CONST robtarget LHP_000:=[[2573.53101,1238.19995,2660.84204],[0.56645757,-0.58473384,0.19941168,-0.54538715],[-1,-1,-1,4],[9E9,9E9,9E9,9E9,9E9,9E9]];
CONST robtarget LHP_005:=[[1933.57397,1076.34998,919.023987],[0.6739808,-0.04561597,0.22679393,-0.70159364],[-1,-1,-1,0],[9E9,9E9,9E9,9E9,9E9,9E9]];
CONST robtarget LHP_010:=[[1910.90503,994.687988,216.904999],[0.7042605,0.08468377,0.09847328,-0.6979605],[-1,-1,-1,0],[9E9,9E9,9E9,9E9,9E9,9E9]];
CONST robtarget LHP_015:=[[1910.89099,994.690002,-385.321991],[0.683501,0.087539785,0.09595496,-0.71830064],[-1,-1,-1,0],[9E9,9E9,9E9,9E9,9E9,9E9]];
CONST robtarget LHP_020:=[[1910.92,803.63,-358.65],[0.683496,0.087554,0.0959515,-0.718305],[-1,-1,-1,0],[9E+09,9E+09,9E+09,9E+09,9E+09,9E+09]];
CONST robtarget LHP_025:=[[1910.97,741.50,-281.66],[0.683494,0.0875455,0.0959486,-0.718307],[-1,-1,-1,0],[9E+09,9E+09,9E+09,9E+09,9E+09,9E+09]];
CONST robtarget LHP_030:=[[1910.91,559.83,-213.69],[0.686476,0.0613746,0.0695917,-0.721208],[-1,-1,-1,0],[9E+09,9E+09,9E+09,9E+09,9E+09,9E+09]];
CONST robtarget LHP_035:=[[1929.33,361.88,-170.13],[0.702471,0.0120548,-0.002609,-0.711605],[-1,0,-1,0],[9E+09,9E+09,9E+09,9E+09,9E+09,9E+09]];
CONST robtarget LHP_040:=[[2007.526,383.55899,-50.7519989],[0.75072795,0.000611088,0.00040383,-0.6606111],[-1,-1,-1,0],[9E9,9E9,9E9,9E9,9E9,9E9]];
CONST robtarget LHP_045:=[[1993.04797,313.046997,-31.7070007],[0.7336252,0.009941696,-0.001285905,-0.67948043],[-1,0,-1,0],[9E9,9E9,9E9,9E9,9E9,9E9]];
CONST robtarget LHP_050:=[[2002.59399,189.292999,-35.1940002],[0.73792726,0.009937888,-0.0012356,-0.67480594],[-1,0,-1,0],[9E9,9E9,9E9,9E9,9E9,9E9]];
CONST robtarget LHP_055:=[[1987.44,-5.82,-69.73],[0.747483,0.000551369,0.000433351,-0.664281],[-1,-1,-1,0],[9E+09,9E+09,9E+09,9E+09,9E+09,9E+09]];
CONST robtarget LHP_060:=[[1929.34,361.89,-170.15],[0.70247,0.0120598,-0.00260928,-0.711607],[-1,0,-1,0],[9E+09,9E+09,9E+09,9E+09,9E+09,9E+09]];
CONST robtarget LHP_065:=[[1910.91,559.85,-213.71],[0.686472,0.0613779,0.0695915,-0.721211],[-1,-1,-1,0],[9E+09,9E+09,9E+09,9E+09,9E+09,9E+09]];
CONST robtarget LHP_070:=[[1769.54,626.69,-228.36],[0.648406,0.063605,0.0595836,-0.756289],[-1,-1,-1,0],[9E+09,9E+09,9E+09,9E+09,9E+09,9E+09]];
CONST robtarget LHP_075:=[[1629.23,373.82,-175.88],[0.60566,0.011527,-0.00436593,-0.795628],[-1,0,-1,0],[9E+09,9E+09,9E+09,9E+09,9E+09,9E+09]];
CONST robtarget LHP_080:=[[1643.37,44.45,-93.67],[0.638426,0.0118697,-0.00343011,-0.769584],[-1,0,-1,0],[9E+09,9E+09,9E+09,9E+09,9E+09,9E+09]];
CONST robtarget LHP_085:=[[1645.79,51.65,-47.78],[0.621544,0.019299,-0.00963586,-0.783082],[-1,0,-1,0],[9E+09,9E+09,9E+09,9E+09,9E+09,9E+09]];
CONST robtarget LHP_090:=[[1652.62,133.53,-52.42],[0.605581,0.0130855,-0.00581803,-0.795655],[-1,0,-1,0],[9E+09,9E+09,9E+09,9E+09,9E+09,9E+09]];
CONST robtarget LHP_095:=[[1617.10803,350.912994,-180.268005],[0.56401443,0.037766688,0.053717423,-0.8231499],[-1,-1,-1,0],[9E9,9E9,9E9,9E9,9E9,9E9]];
CONST robtarget LHP_100:=[[1517.84,635.47,-254.71],[0.565141,-0.00404407,-0.00655324,-0.824958],[-1,0,-1,0],[9E+09,9E+09,9E+09,9E+09,9E+09,9E+09]];
CONST robtarget LHP_105:=[[1647.70,917.36,-357.05],[0.686537,0.012902,0.00966857,-0.726916],[-1,-1,-1,0],[9E+09,9E+09,9E+09,9E+09,9E+09,9E+09]];
CONST robtarget LHP_110:=[[1402.01,954.02,-347.18],[0.618002,-0.00350893,0.00682793,-0.786139],[-1,-1,-1,0],[9E+09,9E+09,9E+09,9E+09,9E+09,9E+09]];
CONST robtarget LHP_115:=[[1380.13,800.38,-344.28],[0.663576,-0.00391562,0.00660285,-0.74807],[-1,-1,-1,0],[9E+09,9E+09,9E+09,9E+09,9E+09,9E+09]];
CONST robtarget LHP_120:=[[1355.05,688.92,-230.68],[0.643458,-0.00406434,0.0069742,-0.765439],[-1,-1,-1,0],[9E+09,9E+09,9E+09,9E+09,9E+09,9E+09]];
CONST robtarget LHP_125:=[[1338.98,616.80,-217.15],[0.641931,-0.00377363,0.00673657,-0.766724],[-1,-1,-1,0],[9E+09,9E+09,9E+09,9E+09,9E+09,9E+09]];
CONST robtarget LHP_130:=[[1328.82,551.60,-198.45],[0.643236,-0.00380631,0.00669098,-0.765629],[-1,-1,-1,0],[9E+09,9E+09,9E+09,9E+09,9E+09,9E+09]];
CONST robtarget LHP_135:=[[1301.19,432.03,-200.08],[0.630965,0.0270779,0.0228783,-0.775001],[-1,-1,-1,0],[9E+09,9E+09,9E+09,9E+09,9E+09,9E+09]];
CONST robtarget LHP_140:=[[1315.22,418.75,-159.95],[0.640955,0.052567,0.0459758,-0.764395],[-1,-1,-1,0],[9E+09,9E+09,9E+09,9E+09,9E+09,9E+09]];
CONST robtarget LHP_145:=[[1314.89,402.01,-58.59],[0.643636,0.0406528,0.0359674,-0.763405],[-1,-1,-1,0],[9E+09,9E+09,9E+09,9E+09,9E+09,9E+09]];
CONST robtarget LHP_150:=[[1314.89,402.00,-58.59],[0.64363700,0.04065100,0.0359677,-0.7634040],[-1,-1,-1,0],[9E+09,9E+09,9E+09,9E+09,9E+09,9E+09]];
CONST robtarget LHP_155:=[[1315.25,418.75,-159.98],[0.640959,0.05257270,0.04597540,-0.7643910],[-1,-1,-1,0],[9E+09,9E+09,9E+09,9E+09,9E+09,9E+09]];
CONST robtarget LHP_160:=[[1301.20,432.03,-200.09],[0.630966,0.0270787,0.0228773,-0.775],[-1,-1,-1,0],[9E+09,9E+09,9E+09,9E+09,9E+09,9E+09]];
CONST robtarget LHP_165:=[[1328.84,551.60,-198.48],[0.643767,-0.00379566,0.00669219,-0.765183],[-1,-1,-1,0],[9E+09,9E+09,9E+09,9E+09,9E+09,9E+09]];
CONST robtarget LHP_170:=[[1356.81,663.69,-214.66],[0.64609,-0.00377796,0.00670482,-0.7632220],[-1,-1,-1,0],[9E+09,9E+09,9E+09,9E+09,9E+09,9E+09]];
CONST robtarget LHP_175:=[[1392.09,854.35,-337.39],[0.646086,-0.00378978,0.00670626,-0.763226],[-1,-1,-1,0],[9E+09,9E+09,9E+09,9E+09,9E+09,9E+09]];
CONST robtarget LHP_180:=[[1392.10,915.32,-339.98],[0.646085,-0.00379686,0.00670629,-0.763227],[-1,-1,-1,0],[9E+09,9E+09,9E+09,9E+09,9E+09,9E+09]];
CONST robtarget LHP_185:=[[1392.13,915.34,-336.92],[0.646086,-0.00378783,0.00670572,-0.763226],[-1,-1,-1,0],[9E+09,9E+09,9E+09,9E+09,9E+09,9E+09]];
CONST robtarget LHP_190:=[[1777.10,396.39,-174.51],[0.778298,0.00338922,-0.00251072,-0.62788],[-1,0,-1,0],[9E+09,9E+09,9E+09,9E+09,9E+09,9E+09]];
CONST robtarget LHP_195:=[[1816.72,397.75,-147.92],[0.816486,0.00152322,-0.000785194,-0.577362],[-1,0,-1,0],[9E+09,9E+09,9E+09,9E+09,9E+09,9E+09]];
CONST robtarget LHP_200:=[[1816.69,397.74,-147.92],[0.816487,0.00151316,-0.000780112,-0.577362],[-1,0,-1,0],[9E+09,9E+09,9E+09,9E+09,9E+09,9E+09]];
CONST robtarget LHP_205:=[[1684.96,400.28,-45.26],[0.59824,-0.000475336,-0.0146536,-0.801183],[-1,0,-1,0],[9E+09,9E+09,9E+09,9E+09,9E+09,9E+09]];
CONST robtarget LHP_210:=[[1517.37,845.68,-347.51],[0.603966,0.0765094,0.0409368,-0.792272],[-1,-1,-1,0],[9E+09,9E+09,9E+09,9E+09,9E+09,9E+09]];
CONST robtarget LHP_215:=[[1614.81,303.29,-114.97],[0.595541,4.37463E-06,7.52158E-05,-0.803325],[-1,-1,-1,0],[9E+09,9E+09,9E+09,9E+09,9E+09,9E+09]];
CONST robtarget LHP_220:=[[1496.10,381.00,-140.90],[0.501832,0.0142883,0.0357857,-0.864106],[-1,-1,-1,0],[9E+09,9E+09,9E+09,9E+09,9E+09,9E+09]];
CONST robtarget LHP_225:=[[1496.16,381.04,-179.37],[0.501836,0.0143261,0.0358019,-0.864103],[-1,-1,-1,0],[9E+09,9E+09,9E+09,9E+09,9E+09,9E+09]];
CONST robtarget LHP_230:=[[1517.37,556.59,-186.35],[0.545787,0.0365786,0.0545327,-0.835347],[-1,-1,-1,0],[9E+09,9E+09,9E+09,9E+09,9E+09,9E+09]];
CONST robtarget LHP_235:=[[1529.66,619.50,-150.47],[0.565262,-0.000227126,0.000165536,-0.824912],[-1,-1,-1,0],[9E+09,9E+09,9E+09,9E+09,9E+09,9E+09]];
CONST robtarget LHP_240:=[[1558.44,796.09,-349.49],[0.583985,0.0684408,0.0319346,-0.808244],[-1,-1,-1,0],[9E+09,9E+09,9E+09,9E+09,9E+09,9E+09]];
CONST robtarget LHP_245:=[[1477.93,985.71,-357.82],[0.551096,0.0897034,0.0519627,-0.827978],[-1,-1,-1,0],[9E+09,9E+09,9E+09,9E+09,9E+09,9E+09]];
CONST robtarget LHP_250:=[[807.86,896.51,-348.98],[0.475989,-0.019585,0.0486327,-0.877887],[-1,-1,-1,0],[9E+09,9E+09,9E+09,9E+09,9E+09,9E+09]];
CONST robtarget LHP_255:=[[807.84,813.89,-348.98],[0.47599,-0.0195894,0.0486332,-0.877887],[-1,-1,-1,0],[9E+09,9E+09,9E+09,9E+09,9E+09,9E+09]];
CONST robtarget LHP_260:=[[798.625,757.187988,-251.093002],[0.47488588,-0.019798715,0.048936285,-0.8784627],[-1,-1,-1,0],[9E9,9E9,9E9,9E9,9E9,9E9]];
CONST robtarget LHP_265:=[[687.672974,377.386993,-182.552002],[0.5034063,-0.04137853,0.03811411,-0.8622165],[-1,-1,-1,0],[9E9,9E9,9E9,9E9,9E9,9E9]];
CONST robtarget LHP_270:=[[796.06,403.61,2.12],[0.54967,-0.0809587,0.0198978,-0.831212],[-1,-1,-1,0],[9E+09,9E+09,9E+09,9E+09,9E+09,9E+09]];
CONST robtarget LHP_275:=[[951.56,404.05,-36.64],[0.666081,-0.0483269,0.018538,-0.744081],[-1,-1,-1,0],[9E+09,9E+09,9E+09,9E+09,9E+09,9E+09]];
CONST robtarget LHP_280:=[[1053.17,384.08,-147.35],[0.741703,0.0276666,0.0554714,-0.667858],[-1,-1,-1,0],[9E+09,9E+09,9E+09,9E+09,9E+09,9E+09]];
CONST robtarget LHP_285:=[[1117.00,437.68,-186.63],[0.764604,0.0628167,0.0737039,-0.637183],[-1,-1,-1,0],[9E+09,9E+09,9E+09,9E+09,9E+09,9E+09]];
CONST robtarget LHP_290:=[[1206.43,437.70,-186.66],[0.808318,0.0679399,0.0690137,-0.580726],[-1,-1,-1,0],[9E+09,9E+09,9E+09,9E+09,9E+09,9E+09]];
CONST robtarget LHP_295:=[[1254.01,306.17,-147.47],[0.819239,0.0692406,0.0677067,-0.565215],[-1,-1,-1,0],[9E+09,9E+09,9E+09,9E+09,9E+09,9E+09]];
CONST robtarget LHP_300:=[[1294.76,251.64,-118.31],[0.839473,0.0657832,0.0563212,-0.536456],[-1,-1,-1,0],[9E+09,9E+09,9E+09,9E+09,9E+09,9E+09]];
CONST robtarget LHP_305:=[[1302.68,268.91,-77.08],[0.850295,0.0194976,0.0312356,-0.525017],[-1,-1,-1,0],[9E+09,9E+09,9E+09,9E+09,9E+09,9E+09]];
CONST robtarget LHP_310:=[[1302.67,268.92,-77.09],[0.850295,0.0194964,0.0312402,-0.525016],[-1,-1,-1,0],[9E+09,9E+09,9E+09,9E+09,9E+09,9E+09]];
CONST robtarget LHP_315:=[[1294.76,251.64,-118.31],[0.839473,0.0657839,0.0563209,-0.536456],[-1,-1,-1,0],[9E+09,9E+09,9E+09,9E+09,9E+09,9E+09]];
CONST robtarget LHP_320:=[[1254.01,306.17,-147.47],[0.819239,0.0692405,0.0677067,-0.565215],[-1,-1,-1,0],[9E+09,9E+09,9E+09,9E+09,9E+09,9E+09]];
CONST robtarget LHP_325:=[[1206.43,437.70,-186.66],[0.808318,0.0679399,0.0690137,-0.580726],[-1,-1,-1,0],[9E+09,9E+09,9E+09,9E+09,9E+09,9E+09]];
CONST robtarget LHP_330:=[[1117.00,437.68,-186.63],[0.764604,0.0628167,0.0737039,-0.637183],[-1,-1,-1,0],[9E+09,9E+09,9E+09,9E+09,9E+09,9E+09]];
CONST robtarget LHP_335:=[[1116.98,404.12,-155.12],[0.767929,0.0632076,0.0733697,-0.633172],[-1,-1,-1,0],[9E+09,9E+09,9E+09,9E+09,9E+09,9E+09]];
CONST robtarget LHP_340:=[[1116.98,404.12,-77.86],[0.763388,0.0288222,0.0341692,-0.644392],[-1,-1,-1,0],[9E+09,9E+09,9E+09,9E+09,9E+09,9E+09]];
CONST robtarget LHP_345:=[[951.56,404.05,-36.63],[0.666079,-0.0483271,0.018537,-0.744083],[-1,-1,-1,0],[9E+09,9E+09,9E+09,9E+09,9E+09,9E+09]];
CONST robtarget LHP_350:=[[863.42,413.34,0.81],[0.590286,-0.0726155,0.0279581,-0.803435],[-1,-1,-1,0],[9E+09,9E+09,9E+09,9E+09,9E+09,9E+09]];
CONST robtarget LHP_355:=[[687.66803,377.371002,-182.531006],[0.5034058,-0.04138605,0.0381097,-0.8622166],[-1,-1,-1,0],[9E9,9E9,9E9,9E9,9E9,9E9]];
CONST robtarget LHP_360:=[[798.580994,757.198975,-251.070007],[0.47486982,-0.019813199,0.04892835,-0.8784715],[-1,-1,-1,0],[9E9,9E9,9E9,9E9,9E9,9E9]];
CONST robtarget LHP_365:=[[961.40,981.11,-456.97],[0.440335,0.0935079,0.0750373,-0.889792],[-1,-1,-1,0],[9E+09,9E+09,9E+09,9E+09,9E+09,9E+09]];
CONST robtarget LHP_370:=[[1477.90,985.72,-357.83],[0.558631,0.0901634,0.0511329,-0.822914],[-1,-1,-1,0],[9E+09,9E+09,9E+09,9E+09,9E+09,9E+09]];
CONST robtarget LHP_375:=[[1538.22,786.86,-339.64],[0.544053,0.0691445,0.0535195,-0.834482],[-1,-1,-1,0],[9E+09,9E+09,9E+09,9E+09,9E+09,9E+09]];
CONST robtarget LHP_380:=[[1502.92,670.32,-266.02],[0.529086,0.0479959,0.0506422,-0.845695],[-1,-1,-1,0],[9E+09,9E+09,9E+09,9E+09,9E+09,9E+09]];
CONST robtarget LHP_385:=[[1496.13,395.81,-167.92],[0.501832,0.0142997,0.0357903,-0.864106],[-1,-1,-1,0],[9E+09,9E+09,9E+09,9E+09,9E+09,9E+09]];
CONST robtarget LHP_390:=[[1515.01,305.29,-41.45],[0.500229,-6.95049E-05,2.93455E-05,-0.865893],[-1,-1,-1,0],[9E+09,9E+09,9E+09,9E+09,9E+09,9E+09]];
CONST robtarget LHP_395:=[[1371.85706,156.694901,-47.4344292],[0.4850808,-0.004593692,-0.00611278,-0.8744359],[-1,0,-1,0],[9E9,9E9,9E9,9E9,9E9,9E9]];
CONST robtarget LHP_400:=[[1371.81006,156.684998,-41.7470016],[0.48507392,-0.004586132,-0.006106427,-0.8744398],[-1,0,-1,0],[9E9,9E9,9E9,9E9,9E9,9E9]];
CONST robtarget LHP_405:=[[1492.72,315.84,-138.22],[0.571745,-0.00395765,-0.00657566,-0.820395],[-1,0,-1,0],[9E+09,9E+09,9E+09,9E+09,9E+09,9E+09]];
CONST robtarget LHP_410:=[[1568.64,542.95,-202.94],[0.571744,-0.00395848,-0.00658119,-0.820396],[-1,0,-1,0],[9E+09,9E+09,9E+09,9E+09,9E+09,9E+09]];
CONST robtarget LHP_415:=[[1568.58,736.45,-284.14],[0.571745,-0.00397095,-0.00657964,-0.820396],[-1,0,-1,0],[9E+09,9E+09,9E+09,9E+09,9E+09,9E+09]];
CONST robtarget LHP_420:=[[1508.30,917.00,-395.22],[0.556499,0.0508994,0.0317793,-0.828678],[-1,-1,-1,0],[9E+09,9E+09,9E+09,9E+09,9E+09,9E+09]];
CONST robtarget LHP_425:=[[1495.25,987.39,-357.83],[0.551104,0.0895725,0.0518729,-0.827992],[-1,-1,-1,0],[9E+09,9E+09,9E+09,9E+09,9E+09,9E+09]];
CONST robtarget LHP_430:=[[1328.35,635.44,-278.20],[0.501405,0.0212305,0.11734,-0.856956],[-1,-1,0,0],[9E+09,9E+09,9E+09,9E+09,9E+09,9E+09]];
CONST robtarget LHP_435:=[[1126.70,526.89,-238.13],[0.384755,0.0646485,0.107006,-0.914513],[-1,-1,0,0],[9E+09,9E+09,9E+09,9E+09,9E+09,9E+09]];
CONST robtarget LHP_440:=[[1126.70,526.87,-238.14],[0.384757,0.0646487,0.107006,-0.914512],[-1,-1,0,0],[9E+09,9E+09,9E+09,9E+09,9E+09,9E+09]];
CONST robtarget LHP_445:=[[1328.35,635.43,-278.21],[0.501406,0.0212292,0.11734,-0.856956],[-1,-1,0,0],[9E+09,9E+09,9E+09,9E+09,9E+09,9E+09]];
CONST robtarget LHP_450:=[[1495.26,987.39,-357.84],[0.551103,0.0895724,0.0518701,-0.827993],[-1,-1,-1,0],[9E+09,9E+09,9E+09,9E+09,9E+09,9E+09]];
CONST robtarget LHP_455:=[[1606.25,805.30,-336.47],[0.591189,0.0705667,0.0504833,-0.801852],[-1,-1,-1,0],[9E+09,9E+09,9E+09,9E+09,9E+09,9E+09]];
CONST robtarget LHP_460:=[[1846.21,646.41,-266.45],[0.66313,0.055392,0.0578373,-0.744207],[-1,-1,-1,0],[9E+09,9E+09,9E+09,9E+09,9E+09,9E+09]];
CONST robtarget LHP_465:=[[1831.93,634.62,-78.38],[0.625946,0.00957367,0.0100376,-0.779743],[-1,-1,-1,0],[9E+09,9E+09,9E+09,9E+09,9E+09,9E+09]];
CONST robtarget LHP_470:=[[1778.25,512.89,-42.92],[0.553639,0.000122695,-2.9028E-05,-0.832757],[-1,-1,-1,0],[9E+09,9E+09,9E+09,9E+09,9E+09,9E+09]];
CONST robtarget LHP_475:=[[1581.22,548.75,-125.86],[0.508525,0.0149425,0.00198371,-0.860915],[-1,0,-1,0],[9E+09,9E+09,9E+09,9E+09,9E+09,9E+09]];
CONST robtarget LHP_480:=[[1526.71,530.36,-111.44],[0.495097,0.0157343,0.00230728,-0.868692],[-1,0,-1,0],[9E+09,9E+09,9E+09,9E+09,9E+09,9E+09]];
CONST robtarget LHP_485:=[[1496.52905,533.620972,-169.427002],[0.5015252,0.014323151,0.035049833,-0.8643141],[-1,-1,-1,0],[9E9,9E9,9E9,9E9,9E9,9E9]];
CONST robtarget LHP_490:=[[1628.88,359.00,-167.42],[0.509965,0.00587853,-0.00326077,-0.860169],[-1,0,-1,0],[9E+09,9E+09,9E+09,9E+09,9E+09,9E+09]];
CONST robtarget LHP_495:=[[1653.10,363.04,-167.43],[0.50985,0.0307676,0.0114918,-0.859636],[-1,0,-1,0],[9E+09,9E+09,9E+09,9E+09,9E+09,9E+09]];
CONST robtarget LHP_500:=[[1734.14,581.56,-229.81],[0.51369,0.0926739,0.046858,-0.851668],[-1,-1,-1,0],[9E+09,9E+09,9E+09,9E+09,9E+09,9E+09]];
CONST robtarget LHP_505:=[[1850.77,754.32,-287.10],[0.562259,0.138379,0.0973397,-0.809469],[-1,-1,-1,0],[9E+09,9E+09,9E+09,9E+09,9E+09,9E+09]];
CONST robtarget LHP_510:=[[1850.71,883.30,-361.37],[0.589549,0.148661,0.155296,-0.778598],[-1,-1,-1,0],[9E+09,9E+09,9E+09,9E+09,9E+09,9E+09]];
CONST robtarget LHP_515:=[[1850.60,911.16,-304.76],[0.610795,0.143869,0.202267,-0.751877],[-1,-1,-1,0],[9E+09,9E+09,9E+09,9E+09,9E+09,9E+09]];
CONST robtarget LHP_520:=[[1845.93,938.54,-187.19],[0.617535,0.126482,0.223985,-0.743292],[-1,-1,-1,0],[9E+09,9E+09,9E+09,9E+09,9E+09,9E+09]];
CONST robtarget LHP_525:=[[1839.91,764.25,251.37],[0.609113,0.0794277,0.135403,-0.777392],[-1,-1,-1,0],[9E+09,9E+09,9E+09,9E+09,9E+09,9E+09]];
CONST robtarget LHP_530:=[[1951.53,815.35,1215.32],[0.610126,-0.0704393,-0.00824645,-0.789124],[-1,0,-1,0],[9E+09,9E+09,9E+09,9E+09,9E+09,9E+09]];
CONST robtarget LHP_535:=[[2438.93,960.39,2235.39],[0.671457,-0.189483,-0.125804,-0.705277],[-1,0,-1,0],[9E+09,9E+09,9E+09,9E+09,9E+09,9E+09]];
!provisorische Punkte fuer SP-Versetzung in Zone2
CONST robtarget LHP_605:=[[1647.70,917.36,-357.05],[0.686537,0.012902,0.00966857,-0.726916],[-1,-1,-1,0],[9E+09,9E+09,9E+09,9E+09,9E+09,9E+09]];
CONST robtarget LHP_610:=[[1610.73,498.12,-174.33],[0.637115,0.00115243,-0.000308458,-0.770768],[-1,0,-1,0],[9E+09,9E+09,9E+09,9E+09,9E+09,9E+09]];
CONST robtarget LHP_620:=[[1777.10,396.39,-174.52],[0.764298,0.00344259,-0.00243544,-0.644849],[-1,0,-1,0],[9E+09,9E+09,9E+09,9E+09,9E+09,9E+09]];
CONST robtarget LHP_625:=[[1816.72,397.75,-147.92],[0.816486,0.00152322,-0.000785194,-0.577362],[-1,0,-1,0],[9E+09,9E+09,9E+09,9E+09,9E+09,9E+09]];
CONST robtarget LHP_630:=[[1816.69,397.74,-147.92],[0.816487,0.00151316,-0.000780112,-0.577362],[-1,0,-1,0],[9E+09,9E+09,9E+09,9E+09,9E+09,9E+09]];
CONST robtarget LHP_635:=[[1517.21,788.33,-328.51],[0.603967,0.0765054,0.0409354,-0.792272],[-1,-1,-1,0],[9E+09,9E+09,9E+09,9E+09,9E+09,9E+09]];
CONST robtarget LHP_600:=[[1990.20,974.03,1486.76],[0.667207,-0.21865,0.214527,-0.678974],[-1,-1,-1,0],[9E+09,9E+09,9E+09,9E+09,9E+09,9E+09]];
! ------------------------------------------------------------
! Unterprogramm:
! Stand
! Daimler AG - Werk Ludwigsfelde
! ------------------------------------------------------------
! ************************************************************
! Kommentar: Achtung
! automatisch generiert!!!!!!!!!!!!!!!!!!
! ************************************************************

! Robotername: 1606R04
! Anlagenbezeichn: Linie 16 Stations-Nr: 1606
! Stand / Version: 04.08.2009 / 1.1
! Name Bearbeiter: Karmann
! Applikationssteuerung: Punktschweissen
! Baumuster: FHL T1 R2


INIT_SW_BASE;

WKZ_1_AUFNEHMEN;

MoveJ ToolHome1,vSchnell,fine,nomtcp1;

MoveJ LHP_000,vSchnell,fine,nomtcp1\WObj:=BS_1606_1A;

Vorhub\auf;

ABL 2\ABL_WAIT;
ABL 10\ABL_SET;

!1606R04_1606R06
KOLLISION_ZONE 2\Anfrage;
!1606R04_1606R06
KOLLISION_ZONE 7\Anfrage;
!1606R04_1606R06
KOLLISION_ZONE 9\Anfrage;

MoveJ LHP_600, vSchnell, fine, nomtcp1\WObj:=BS_1606_1A;

!
! robic dojazd
!
WaitUntil FALSE;

MoveJ LHP_165,vSchnell,z100,nomtcp1\WObj:=BS_1606_1A;
MoveJ LHP_160,vSchnell,z1,nomtcp1\WObj:=BS_1606_1A;
MoveJ LHP_155,vSchnell,z1,nomtcp1\WObj:=BS_1606_1A;
MoveJ LHP_150,vSchnell,z1,nomtcp1\WObj:=BS_1606_1A;

SpotL G0216190478BP20\VFO:=210,vSpot,nomtcp1\WObj:=BS_1606_1A;
SpotL G0216190582BP20\VFO:=210,vSpot,nomtcp1\WObj:=BS_1606_1A;

MoveJ LHP_120,vSchnell,z100,nomtcp1\WObj:=BS_1606_1A;
MoveJ LHP_125,vSchnell,z100,nomtcp1\WObj:=BS_1606_1A;

SpotL G0216190492BP20\VFO:=210\Vorhub_Auf,vSpot,nomtcp1\WObj:=BS_1606_1A;

KOLLISION_ZONE 2\Freigabe;

!
! zrobic dojazd
!
WaitUntil FALSE;

MoveJ LHP_480,vSchnell,z100,nomtcp1\WObj:=BS_1606_1A;

SpotL G0216190576BP20\VFO:=210,vSpot,nomtcp1\WObj:=BS_1606_1A;
SpotL G0213198812BP20\VFO:=210\Vorhub_Auf,vSpot,nomtcp1\WObj:=BS_1606_1A;

MoveJ LHP_485,vSchnell,z100,nomtcp1\WObj:=BS_1606_1A;

!
! zrobic dojazd
!
WaitUntil FALSE;

SpotL G0213198810BP20\VFO:=210,vSpot,nomtcp1\WObj:=BS_1606_1A;
SpotL G0213198808BP20\VFO:=210,vSpot,nomtcp1\WObj:=BS_1606_1A;
SpotL G0216021648BP20\VFO:=210,vSpot,nomtcp1\WObj:=BS_1606_1A;
SpotL G0216021650BP20\VFO:=210,vSpot,nomtcp1\WObj:=BS_1606_1A;

MoveJ LHP_470,vSchnell,fine,nomtcp1\WObj:=BS_1606_1A;

SpotL G0216021652BP20\VFO:=210,vSpot,nomtcp1\WObj:=BS_1606_1A;

!
! zrobic dojazd
!
WaitUntil FALSE;

MoveJ LHP_620,vSchnell,z100,nomtcp1\WObj:=BS_1606_1A;
MoveJ LHP_625,vSchnell,z100,nomtcp1\WObj:=BS_1606_1A;

SpotL G0216021802BP20\VFO:=210\Vorhub_Auf,vSpot,nomtcp1\WObj:=BS_1606_1A;

MoveJ LHP_630,vSchnell,z100,nomtcp1\WObj:=BS_1606_1A;

!
! zrobic dojazd
!
WaitUntil FALSE;

MoveJ LHP_025,vSchnell,z100,nomtcp1\WObj:=BS_1606_1A;
MoveJ LHP_030,vSchnell,z100,nomtcp1\WObj:=BS_1606_1A;
MoveJ LHP_035,vSchnell,z100,nomtcp1\WObj:=BS_1606_1A;

SpotL G0216021800BP20\VFO:=210,vSpot,nomtcp1\WObj:=BS_1606_1A;
SpotL G0216021798BP20\VFO:=210\Vorhub_Auf,vSpot,nomtcp1\WObj:=BS_1606_1A;

!
! zrobic dojazd
!
WaitUntil FALSE;

SpotL G0216021654BP20\VFO:=210,vSpot,nomtcp1\WObj:=BS_1606_1A;
SpotL G0216190440BP20\VFO:=210,vSpot,nomtcp1\WObj:=BS_1606_1A;
SpotL G0216190438BP20\VFO:=210,vSpot,nomtcp1\WObj:=BS_1606_1A;

MoveJ LHP_455,vSchnell,z100,nomtcp1\WObj:=BS_1606_1A;
MoveJ LHP_460,vSchnell,z100,nomtcp1\WObj:=BS_1606_1A;
MoveJ LHP_465,vSchnell,z100,nomtcp1\WObj:=BS_1606_1A;

SpotL G0216190436BP20\VFO:=210\Vorhub_Auf,vSpot,nomtcp1\WObj:=BS_1606_1A;

!
! zrobic dojazd
!
WaitUntil FALSE;

MoveJ LHP_475,vSchnell,z100,nomtcp1\WObj:=BS_1606_1A;

SpotL G0216190434BP20\VFO:=210,vSpot,nomtcp1\WObj:=BS_1606_1A;
SpotL G0216190432BP20\VFO:=210,vSpot,nomtcp1\WObj:=BS_1606_1A;
SpotL G0216190430BP20\VFO:=210,vSpot,nomtcp1\WObj:=BS_1606_1A;

MoveJ LHP_450,vSchnell,z100,nomtcp1\WObj:=BS_1606_1A;

SpotL G0216190428BP20\VFO:=210\Vorhub_Auf,vSpot,nomtcp1\WObj:=BS_1606_1A;

!
! zrobic dojazd
!
WaitUntil FALSE;

MoveJ LHP_230,vSchnell,z100,nomtcp1\WObj:=BS_1606_1A;

SpotL G0216190446BP20\VFO:=210\Vorhub_Auf,vSpot,nomtcp1\WObj:=BS_1606_1A;

MoveJ LHP_235,vSchnell,z100,nomtcp1\WObj:=BS_1606_1A;
MoveJ LHP_610,vSchnell,fine,nomtcp1\WObj:=BS_1606_1A;

!
! zrobic dojazd
!
WaitUntil FALSE;

MoveJ LHP_250,vSchnell,fine,nomtcp1\WObj:=BS_1606_1A;

!1606R04_1606R06
KOLLISION_ZONE 1\Anfrage;
!1606R04_1606R06
KOLLISION_ZONE 6\Anfrage;

MoveJ LHP_255,vSchnell,z100,nomtcp1\WObj:=BS_1606_1A;
MoveJ LHP_260,vSchnell,z100,nomtcp1\WObj:=BS_1606_1A;
MoveJ LHP_265,vSchnell,z100,nomtcp1\WObj:=BS_1606_1A;
MoveJ LHP_270,vSchnell,z100,nomtcp1\WObj:=BS_1606_1A;
MoveJ LHP_275,vSchnell,z100,nomtcp1\WObj:=BS_1606_1A;
MoveJ LHP_280,vSchnell,z100,nomtcp1\WObj:=BS_1606_1A;
MoveL LHP_285,vSchnell,z5,nomtcp1\WObj:=BS_1606_1A;
MoveL LHP_290,vSchnell,z5,nomtcp1\WObj:=BS_1606_1A;
MoveL LHP_295,vSchnell,z5,nomtcp1\WObj:=BS_1606_1A;
MoveL LHP_300,vSchnell,z5,nomtcp1\WObj:=BS_1606_1A;
MoveL LHP_305,vSchnell,z5,nomtcp1\WObj:=BS_1606_1A;

SpotL G0216190480BP20\VFO:=210\Vorhub_Auf, vSpot, nomtcp1\WObj:=BS_1606_1A;

MoveL LHP_310,vSchnell,z5,nomtcp1\WObj:=BS_1606_1A;
MoveL LHP_315,vSchnell,z5,nomtcp1\WObj:=BS_1606_1A;
MoveL LHP_320,vSchnell,z5,nomtcp1\WObj:=BS_1606_1A;
MoveL LHP_325,vSchnell,z5,nomtcp1\WObj:=BS_1606_1A;
MoveL LHP_330,vSchnell,z5,nomtcp1\WObj:=BS_1606_1A;
MoveL LHP_335,vSchnell,z5,nomtcp1\WObj:=BS_1606_1A;
MoveL LHP_340,vSchnell,z5,nomtcp1\WObj:=BS_1606_1A;

SpotL G0216022394BP20\VFO:=210\Vorhub_Auf,vSpot,nomtcp1\WObj:=BS_1606_1A;

MoveJ LHP_345,vSchnell,fine,nomtcp1\WObj:=BS_1606_1A;
MoveJ LHP_350,vSchnell,z100,nomtcp1\WObj:=BS_1606_1A;

SpotL G0216022386BP20\VFO:=210,vSpot,nomtcp1\WObj:=BS_1606_1A;

!1606R04_1606R06
KOLLISION_ZONE 6\Freigabe;

SpotL G0216047033BP20\VFO:=210,vSpot,nomtcp1\WObj:=BS_1606_1A;
SpotL G0216047032BP20\VFO:=210\Vorhub_Auf,vSpot,nomtcp1\WObj:=BS_1606_1A;

MoveJ LHP_355,vSchnell,z100,nomtcp1\WObj:=BS_1606_1A;
MoveJ LHP_360,vSchnell,z100,nomtcp1\WObj:=BS_1606_1A;
MoveJ LHP_365,vSchnell,z100,nomtcp1\WObj:=BS_1606_1A;
MoveJ LHP_370,vSchnell,z100,nomtcp1\WObj:=BS_1606_1A;
!
! zrobic dojazd
!
WaitUntil FALSE;

MoveJ LHP_420,vSchnell,z100,nomtcp1\WObj:=BS_1606_1A;
MoveJ LHP_425,vSchnell,z100,nomtcp1\WObj:=BS_1606_1A;
MoveJ LHP_430,vSchnell,z100,nomtcp1\WObj:=BS_1606_1A;
MoveJ LHP_435,vSchnell,z100,nomtcp1\WObj:=BS_1606_1A;

SpotL G0216047028BP20\VFO:=210,vSpot,nomtcp1\WObj:=BS_1606_1A;
SpotL G0216047029BP20\VFO:=210,vSpot,nomtcp1\WObj:=BS_1606_1A;
SpotL G0216022368BP20\VFO:=210,vSpot,nomtcp1\WObj:=BS_1606_1A;
SpotL G0216022370BP20\VFO:=210\Vorhub_Auf,vSpot,nomtcp1\WObj:=BS_1606_1A;

MoveJ LHP_440,vSchnell,z100,nomtcp1\WObj:=BS_1606_1A;

!
! zrobic dojazd
!
waituntil FALSE;

MoveJ LHP_040,vSchnell,z100,nomtcp1\WObj:=BS_1606_1A;

SpotL G0216190516BP20\VFO:=210,vSpot,nomtcp1\WObj:=BS_1606_1A;

MoveJ LHP_045,vSchnell,z100,nomtcp1\WObj:=BS_1606_1A;

KOLLISION_ZONE 1\Freigabe;
KOLLISION_ZONE 7\Freigabe;
KOLLISION_ZONE 8\Anfrage;

SpotL G0216190518BP20\VFO:=210,vSpot,nomtcp1\WObj:=BS_1606_1A;
SpotL G0216190520BP20\VFO:=210,vSpot,nomtcp1\WObj:=BS_1606_1A;

MoveJ LHP_050,vSchnell,z100,nomtcp1\WObj:=BS_1606_1A;

SpotL G0216190522BP20\VFO:=210,vSpot,nomtcp1\WObj:=BS_1606_1A;
SpotL G0216190524BP20\VFO:=210,vSpot,nomtcp1\WObj:=BS_1606_1A;

!1606R04_1606R03
KOLLISION_ZONE 4\Anfrage;

SpotL G0216190526BP20\VFO:=210,vSpot,nomtcp1\WObj:=BS_1606_1A;
SpotL G0216190528BP20\VFO:=210\Vorhub_Auf, vSpot, nomtcp1\WObj:=BS_1606_1A;

MoveJ LHP_055,vSchnell,z100,nomtcp1\WObj:=BS_1606_1A;
MoveJ LHP_060,vSchnell,z100,nomtcp1\WObj:=BS_1606_1A;
MoveJ LHP_065,vSchnell,z100,nomtcp1\WObj:=BS_1606_1A;
MoveJ LHP_070,vSchnell,z100,nomtcp1\WObj:=BS_1606_1A;
MoveJ LHP_075,vSchnell,z100,nomtcp1\WObj:=BS_1606_1A;
MoveJ LHP_080,vSchnell,z100,nomtcp1\WObj:=BS_1606_1A;

SpotL G0216190508BP20\VFO:=210,vSpot,nomtcp1\WObj:=BS_1606_1A;

MoveJ LHP_085,vSchnell,z100,nomtcp1\WObj:=BS_1606_1A;
MoveJ LHP_090,vSchnell,z100,nomtcp1\WObj:=BS_1606_1A;

SpotL G0216190500BP20\VFO:=210,vSpot,nomtcp1\WObj:=BS_1606_1A;
SpotL G0216190506BP20\VFO:=210,vSpot,nomtcp1\WObj:=BS_1606_1A;

!
! zrobic dojazd
!
WaitUntil FALSE;

MoveJ LHP_385,vSchnell,z100,nomtcp1\WObj:=BS_1606_1A;
MoveJ LHP_390,vSchnell,fine,nomtcp1\WObj:=BS_1606_1A;

!1606R04_1606R06
KOLLISION_ZONE 7\Freigabe;

SpotL G0216190498BP20\VFO:=210,vSpot,nomtcp1\WObj:=BS_1606_1A;

MoveJ LHP_395,vSchnell,z100,nomtcp1\WObj:=BS_1606_1A;

SpotL G0216190488BP20\VFO:=210,vSpot,nomtcp1\WObj:=BS_1606_1A;

MoveJ LHP_400,vSchnell,z100,nomtcp1\WObj:=BS_1606_1A;

SpotL G0216190496BP20\VFO:=210,vSpot,nomtcp1\WObj:=BS_1606_1A;
SpotL G0216190494BP20\VFO:=210\Vorhub_Auf,vSpot,nomtcp1\WObj:=BS_1606_1A;

MoveJ LHP_405,vSchnell,z100,nomtcp1\WObj:=BS_1606_1A;

!
! zrobic dojazd
!
WaitUntil FALSE;

SpotL G0216190502BP20\VFO:=210\Vorhub_Auf,vSpot,nomtcp1\WObj:=BS_1606_1A;

MoveJ LHP_215, vSchnell, z100, nomtcp1\WObj:=BS_1606_1A;
MoveJ LHP_220, vSchnell, z100, nomtcp1\WObj:=BS_1606_1A;

KOLLISION_ZONE 8\Freigabe;

SpotL G0213198814BP20\VFO:=210\Vorhub_Auf,vSpot,nomtcp1\WObj:=BS_1606_1A;

MoveJ LHP_225,vSchnell,z100,nomtcp1\WObj:=BS_1606_1A;

!
! zrobic dojazd
!
WaitUntil FALSE;

SpotL G0213198816BP20\VFO:=210,vSpot,nomtcp1\WObj:=BS_1606_1A;
SpotL G0213198818BP20\VFO:=210\Vorhub_Auf,vSpot,nomtcp1\WObj:=BS_1606_1A;

MoveJ LHP_495,vSchnell,z100,nomtcp1\WObj:=BS_1606_1A;
MoveJ LHP_500,vSchnell,z10,nomtcp1\WObj:=BS_1606_1A;
MoveJ LHP_505,vSchnell,z5,nomtcp1\WObj:=BS_1606_1A;

!
! zrobic dojazd
!
WaitUntil FALSE;

MoveJ LHP_205,vSchnell,z100,nomtcp1\WObj:=BS_1606_1A;

SpotL G0216021806BP20\VFO:=210,vSpot,nomtcp1\WObj:=BS_1606_1A;
SpotL G0216021804BP20\VFO:=210\Vorhub_Auf,vSpot,nomtcp1\WObj:=BS_1606_1A;


!1606R04_1606R06
KOLLISION_ZONE 1\Freigabe;

MoveJ LHP_535, vSchnell, z100, nomtcp1\WObj:=BS_1606_1A;

MoveJ ToolHome1,vSchnell,fine,nomtcp1;


ABL 254\ABL_WAIT;
ABL 255\ABL_SET;

!1606R04_1606R06
KOLLISION_ZONE 9\Freigabe;

ENDPROC







PROC swp_223500_0_st1606_1()

CONST robtarget LHP_000:=[[2573.53101,1238.19995,2660.84204],[0.56645757,-0.58473384,0.19941168,-0.54538715],[-1,-1,-1,4],[9E9,9E9,9E9,9E9,9E9,9E9]];
CONST robtarget LHP_005:=[[1933.57397,1076.34998,919.023987],[0.6739808,-0.04561597,0.22679393,-0.70159364],[-1,-1,-1,0],[9E9,9E9,9E9,9E9,9E9,9E9]];
CONST robtarget LHP_010:=[[1910.90503,994.687988,216.904999],[0.7042605,0.08468377,0.09847328,-0.6979605],[-1,-1,-1,0],[9E9,9E9,9E9,9E9,9E9,9E9]];
CONST robtarget LHP_015:=[[1910.89099,994.690002,-385.321991],[0.683501,0.087539785,0.09595496,-0.71830064],[-1,-1,-1,0],[9E9,9E9,9E9,9E9,9E9,9E9]];
CONST robtarget LHP_020:=[[1910.92,803.63,-358.65],[0.683496,0.087554,0.0959515,-0.718305],[-1,-1,-1,0],[9E+09,9E+09,9E+09,9E+09,9E+09,9E+09]];
CONST robtarget LHP_025:=[[1910.97,741.50,-281.66],[0.683494,0.0875455,0.0959486,-0.718307],[-1,-1,-1,0],[9E+09,9E+09,9E+09,9E+09,9E+09,9E+09]];
CONST robtarget LHP_030:=[[1910.91,559.83,-213.69],[0.686476,0.0613746,0.0695917,-0.721208],[-1,-1,-1,0],[9E+09,9E+09,9E+09,9E+09,9E+09,9E+09]];
CONST robtarget LHP_035:=[[1929.33,361.88,-170.13],[0.702471,0.0120548,-0.002609,-0.711605],[-1,0,-1,0],[9E+09,9E+09,9E+09,9E+09,9E+09,9E+09]];
CONST robtarget LHP_040:=[[2007.526,383.55899,-50.7519989],[0.75072795,0.000611088,0.00040383,-0.6606111],[-1,-1,-1,0],[9E9,9E9,9E9,9E9,9E9,9E9]];
CONST robtarget LHP_045:=[[1993.04797,313.046997,-31.7070007],[0.7336252,0.009941696,-0.001285905,-0.67948043],[-1,0,-1,0],[9E9,9E9,9E9,9E9,9E9,9E9]];
CONST robtarget LHP_050:=[[2002.59399,189.292999,-35.1940002],[0.73792726,0.009937888,-0.0012356,-0.67480594],[-1,0,-1,0],[9E9,9E9,9E9,9E9,9E9,9E9]];
CONST robtarget LHP_055:=[[1987.44,-5.82,-69.73],[0.747483,0.000551369,0.000433351,-0.664281],[-1,-1,-1,0],[9E+09,9E+09,9E+09,9E+09,9E+09,9E+09]];
CONST robtarget LHP_060:=[[1929.34,361.89,-170.15],[0.70247,0.0120598,-0.00260928,-0.711607],[-1,0,-1,0],[9E+09,9E+09,9E+09,9E+09,9E+09,9E+09]];
CONST robtarget LHP_065:=[[1910.91,559.85,-213.71],[0.686472,0.0613779,0.0695915,-0.721211],[-1,-1,-1,0],[9E+09,9E+09,9E+09,9E+09,9E+09,9E+09]];
CONST robtarget LHP_070:=[[1769.54,626.69,-228.36],[0.648406,0.063605,0.0595836,-0.756289],[-1,-1,-1,0],[9E+09,9E+09,9E+09,9E+09,9E+09,9E+09]];
CONST robtarget LHP_075:=[[1629.23,373.82,-175.88],[0.60566,0.011527,-0.00436593,-0.795628],[-1,0,-1,0],[9E+09,9E+09,9E+09,9E+09,9E+09,9E+09]];
CONST robtarget LHP_080:=[[1643.37,44.45,-93.67],[0.638426,0.0118697,-0.00343011,-0.769584],[-1,0,-1,0],[9E+09,9E+09,9E+09,9E+09,9E+09,9E+09]];
CONST robtarget LHP_085:=[[1645.79,51.65,-47.78],[0.621544,0.019299,-0.00963586,-0.783082],[-1,0,-1,0],[9E+09,9E+09,9E+09,9E+09,9E+09,9E+09]];
CONST robtarget LHP_090:=[[1652.62,133.53,-52.42],[0.605581,0.0130855,-0.00581803,-0.795655],[-1,0,-1,0],[9E+09,9E+09,9E+09,9E+09,9E+09,9E+09]];
CONST robtarget LHP_095:=[[1617.10803,350.912994,-180.268005],[0.56401443,0.037766688,0.053717423,-0.8231499],[-1,-1,-1,0],[9E9,9E9,9E9,9E9,9E9,9E9]];
CONST robtarget LHP_100:=[[1517.84,635.47,-254.71],[0.565141,-0.00404407,-0.00655324,-0.824958],[-1,0,-1,0],[9E+09,9E+09,9E+09,9E+09,9E+09,9E+09]];
CONST robtarget LHP_105:=[[1647.70,917.36,-357.05],[0.686537,0.012902,0.00966857,-0.726916],[-1,-1,-1,0],[9E+09,9E+09,9E+09,9E+09,9E+09,9E+09]];
CONST robtarget LHP_110:=[[1402.01,954.02,-347.18],[0.618002,-0.00350893,0.00682793,-0.786139],[-1,-1,-1,0],[9E+09,9E+09,9E+09,9E+09,9E+09,9E+09]];
CONST robtarget LHP_115:=[[1380.13,800.38,-344.28],[0.663576,-0.00391562,0.00660285,-0.74807],[-1,-1,-1,0],[9E+09,9E+09,9E+09,9E+09,9E+09,9E+09]];
CONST robtarget LHP_120:=[[1355.05,688.92,-230.68],[0.643458,-0.00406434,0.0069742,-0.765439],[-1,-1,-1,0],[9E+09,9E+09,9E+09,9E+09,9E+09,9E+09]];
CONST robtarget LHP_125:=[[1338.98,616.80,-217.15],[0.641931,-0.00377363,0.00673657,-0.766724],[-1,-1,-1,0],[9E+09,9E+09,9E+09,9E+09,9E+09,9E+09]];
CONST robtarget LHP_130:=[[1328.82,551.60,-198.45],[0.643236,-0.00380631,0.00669098,-0.765629],[-1,-1,-1,0],[9E+09,9E+09,9E+09,9E+09,9E+09,9E+09]];
CONST robtarget LHP_135:=[[1301.19,432.03,-200.08],[0.630965,0.0270779,0.0228783,-0.775001],[-1,-1,-1,0],[9E+09,9E+09,9E+09,9E+09,9E+09,9E+09]];
CONST robtarget LHP_140:=[[1315.22,418.75,-159.95],[0.640955,0.052567,0.0459758,-0.764395],[-1,-1,-1,0],[9E+09,9E+09,9E+09,9E+09,9E+09,9E+09]];
CONST robtarget LHP_145:=[[1314.89,402.01,-58.59],[0.643636,0.0406528,0.0359674,-0.763405],[-1,-1,-1,0],[9E+09,9E+09,9E+09,9E+09,9E+09,9E+09]];
CONST robtarget LHP_150:=[[1314.89,402.00,-58.59],[0.64363700,0.04065100,0.0359677,-0.7634040],[-1,-1,-1,0],[9E+09,9E+09,9E+09,9E+09,9E+09,9E+09]];
CONST robtarget LHP_155:=[[1315.25,418.75,-159.98],[0.640959,0.05257270,0.04597540,-0.7643910],[-1,-1,-1,0],[9E+09,9E+09,9E+09,9E+09,9E+09,9E+09]];
CONST robtarget LHP_160:=[[1301.20,432.03,-200.09],[0.630966,0.0270787,0.0228773,-0.775],[-1,-1,-1,0],[9E+09,9E+09,9E+09,9E+09,9E+09,9E+09]];
CONST robtarget LHP_165:=[[1328.84,551.60,-198.48],[0.643767,-0.00379566,0.00669219,-0.765183],[-1,-1,-1,0],[9E+09,9E+09,9E+09,9E+09,9E+09,9E+09]];
CONST robtarget LHP_170:=[[1356.81,663.69,-214.66],[0.64609,-0.00377796,0.00670482,-0.7632220],[-1,-1,-1,0],[9E+09,9E+09,9E+09,9E+09,9E+09,9E+09]];
CONST robtarget LHP_175:=[[1392.09,854.35,-337.39],[0.646086,-0.00378978,0.00670626,-0.763226],[-1,-1,-1,0],[9E+09,9E+09,9E+09,9E+09,9E+09,9E+09]];
CONST robtarget LHP_180:=[[1392.10,915.32,-339.98],[0.646085,-0.00379686,0.00670629,-0.763227],[-1,-1,-1,0],[9E+09,9E+09,9E+09,9E+09,9E+09,9E+09]];
CONST robtarget LHP_185:=[[1392.13,915.34,-336.92],[0.646086,-0.00378783,0.00670572,-0.763226],[-1,-1,-1,0],[9E+09,9E+09,9E+09,9E+09,9E+09,9E+09]];
CONST robtarget LHP_190:=[[1777.10,396.39,-174.51],[0.778298,0.00338922,-0.00251072,-0.62788],[-1,0,-1,0],[9E+09,9E+09,9E+09,9E+09,9E+09,9E+09]];
CONST robtarget LHP_195:=[[1816.72,397.75,-147.92],[0.816486,0.00152322,-0.000785194,-0.577362],[-1,0,-1,0],[9E+09,9E+09,9E+09,9E+09,9E+09,9E+09]];
CONST robtarget LHP_200:=[[1816.69,397.74,-147.92],[0.816487,0.00151316,-0.000780112,-0.577362],[-1,0,-1,0],[9E+09,9E+09,9E+09,9E+09,9E+09,9E+09]];
CONST robtarget LHP_205:=[[1684.97,400.31,-52.05],[0.598238,-0.000466613,-0.0146497,-0.801185],[-1,0,-1,0],[9E+09,9E+09,9E+09,9E+09,9E+09,9E+09]];
CONST robtarget LHP_210:=[[1517.37,845.68,-347.51],[0.603966,0.0765094,0.0409368,-0.792272],[-1,-1,-1,0],[9E+09,9E+09,9E+09,9E+09,9E+09,9E+09]];
CONST robtarget LHP_215:=[[1614.81,303.29,-114.97],[0.595541,4.37463E-06,7.52158E-05,-0.803325],[-1,-1,-1,0],[9E+09,9E+09,9E+09,9E+09,9E+09,9E+09]];
CONST robtarget LHP_220:=[[1496.10,381.00,-140.90],[0.501832,0.0142883,0.0357857,-0.864106],[-1,-1,-1,0],[9E+09,9E+09,9E+09,9E+09,9E+09,9E+09]];
CONST robtarget LHP_225:=[[1496.16,381.04,-179.37],[0.501836,0.0143261,0.0358019,-0.864103],[-1,-1,-1,0],[9E+09,9E+09,9E+09,9E+09,9E+09,9E+09]];
CONST robtarget LHP_230:=[[1517.37,556.59,-186.35],[0.545787,0.0365786,0.0545327,-0.835347],[-1,-1,-1,0],[9E+09,9E+09,9E+09,9E+09,9E+09,9E+09]];
CONST robtarget LHP_235:=[[1529.66,619.50,-150.47],[0.565262,-0.000227126,0.000165536,-0.824912],[-1,-1,-1,0],[9E+09,9E+09,9E+09,9E+09,9E+09,9E+09]];
CONST robtarget LHP_240:=[[1558.44,796.09,-349.49],[0.583985,0.0684408,0.0319346,-0.808244],[-1,-1,-1,0],[9E+09,9E+09,9E+09,9E+09,9E+09,9E+09]];
CONST robtarget LHP_245:=[[1477.93,985.71,-357.82],[0.551096,0.0897034,0.0519627,-0.827978],[-1,-1,-1,0],[9E+09,9E+09,9E+09,9E+09,9E+09,9E+09]];
CONST robtarget LHP_250:=[[807.86,896.51,-348.98],[0.475989,-0.019585,0.0486327,-0.877887],[-1,-1,-1,0],[9E+09,9E+09,9E+09,9E+09,9E+09,9E+09]];
CONST robtarget LHP_255:=[[807.84,813.89,-348.98],[0.47599,-0.0195894,0.0486332,-0.877887],[-1,-1,-1,0],[9E+09,9E+09,9E+09,9E+09,9E+09,9E+09]];
CONST robtarget LHP_260:=[[798.625,757.187988,-251.093002],[0.47488588,-0.019798715,0.048936285,-0.8784627],[-1,-1,-1,0],[9E9,9E9,9E9,9E9,9E9,9E9]];
CONST robtarget LHP_265:=[[687.672974,377.386993,-182.552002],[0.5034063,-0.04137853,0.03811411,-0.8622165],[-1,-1,-1,0],[9E9,9E9,9E9,9E9,9E9,9E9]];
CONST robtarget LHP_270:=[[796.06,403.61,2.12],[0.54967,-0.0809587,0.0198978,-0.831212],[-1,-1,-1,0],[9E+09,9E+09,9E+09,9E+09,9E+09,9E+09]];
CONST robtarget LHP_275:=[[951.56,404.05,-36.64],[0.666081,-0.0483269,0.018538,-0.744081],[-1,-1,-1,0],[9E+09,9E+09,9E+09,9E+09,9E+09,9E+09]];
CONST robtarget LHP_280:=[[1053.17,384.08,-147.35],[0.741703,0.0276666,0.0554714,-0.667858],[-1,-1,-1,0],[9E+09,9E+09,9E+09,9E+09,9E+09,9E+09]];
CONST robtarget LHP_285:=[[1117.00,437.68,-186.63],[0.764604,0.0628167,0.0737039,-0.637183],[-1,-1,-1,0],[9E+09,9E+09,9E+09,9E+09,9E+09,9E+09]];
CONST robtarget LHP_290:=[[1206.43,437.70,-186.66],[0.808318,0.0679399,0.0690137,-0.580726],[-1,-1,-1,0],[9E+09,9E+09,9E+09,9E+09,9E+09,9E+09]];
CONST robtarget LHP_295:=[[1254.01,306.17,-147.47],[0.819239,0.0692406,0.0677067,-0.565215],[-1,-1,-1,0],[9E+09,9E+09,9E+09,9E+09,9E+09,9E+09]];
CONST robtarget LHP_300:=[[1294.76,251.64,-118.31],[0.839473,0.0657832,0.0563212,-0.536456],[-1,-1,-1,0],[9E+09,9E+09,9E+09,9E+09,9E+09,9E+09]];
CONST robtarget LHP_305:=[[1302.68,268.91,-77.08],[0.850295,0.0194976,0.0312356,-0.525017],[-1,-1,-1,0],[9E+09,9E+09,9E+09,9E+09,9E+09,9E+09]];
CONST robtarget LHP_310:=[[1302.67,268.92,-77.09],[0.850295,0.0194964,0.0312402,-0.525016],[-1,-1,-1,0],[9E+09,9E+09,9E+09,9E+09,9E+09,9E+09]];
CONST robtarget LHP_315:=[[1294.76,251.64,-118.31],[0.839473,0.0657839,0.0563209,-0.536456],[-1,-1,-1,0],[9E+09,9E+09,9E+09,9E+09,9E+09,9E+09]];
CONST robtarget LHP_320:=[[1254.01,306.17,-147.47],[0.819239,0.0692405,0.0677067,-0.565215],[-1,-1,-1,0],[9E+09,9E+09,9E+09,9E+09,9E+09,9E+09]];
CONST robtarget LHP_325:=[[1206.43,437.70,-186.66],[0.808318,0.0679399,0.0690137,-0.580726],[-1,-1,-1,0],[9E+09,9E+09,9E+09,9E+09,9E+09,9E+09]];
CONST robtarget LHP_330:=[[1117.00,437.68,-186.63],[0.764604,0.0628167,0.0737039,-0.637183],[-1,-1,-1,0],[9E+09,9E+09,9E+09,9E+09,9E+09,9E+09]];
CONST robtarget LHP_335:=[[1116.98,404.12,-155.12],[0.767929,0.0632076,0.0733697,-0.633172],[-1,-1,-1,0],[9E+09,9E+09,9E+09,9E+09,9E+09,9E+09]];
CONST robtarget LHP_340:=[[1116.98,404.12,-77.86],[0.763388,0.0288222,0.0341692,-0.644392],[-1,-1,-1,0],[9E+09,9E+09,9E+09,9E+09,9E+09,9E+09]];
CONST robtarget LHP_345:=[[951.56,404.05,-36.63],[0.666079,-0.0483271,0.018537,-0.744083],[-1,-1,-1,0],[9E+09,9E+09,9E+09,9E+09,9E+09,9E+09]];
CONST robtarget LHP_350:=[[863.42,413.34,0.81],[0.590286,-0.0726155,0.0279581,-0.803435],[-1,-1,-1,0],[9E+09,9E+09,9E+09,9E+09,9E+09,9E+09]];
CONST robtarget LHP_355:=[[687.66803,377.371002,-182.531006],[0.5034058,-0.04138605,0.0381097,-0.8622166],[-1,-1,-1,0],[9E9,9E9,9E9,9E9,9E9,9E9]];
CONST robtarget LHP_360:=[[798.580994,757.198975,-251.070007],[0.47486982,-0.019813199,0.04892835,-0.8784715],[-1,-1,-1,0],[9E9,9E9,9E9,9E9,9E9,9E9]];
CONST robtarget LHP_365:=[[961.40,981.11,-456.97],[0.440335,0.0935079,0.0750373,-0.889792],[-1,-1,-1,0],[9E+09,9E+09,9E+09,9E+09,9E+09,9E+09]];
CONST robtarget LHP_370:=[[1477.90,985.72,-357.83],[0.558631,0.0901634,0.0511329,-0.822914],[-1,-1,-1,0],[9E+09,9E+09,9E+09,9E+09,9E+09,9E+09]];
CONST robtarget LHP_375:=[[1538.22,786.86,-339.64],[0.544053,0.0691445,0.0535195,-0.834482],[-1,-1,-1,0],[9E+09,9E+09,9E+09,9E+09,9E+09,9E+09]];
CONST robtarget LHP_380:=[[1502.92,670.32,-266.02],[0.529086,0.0479959,0.0506422,-0.845695],[-1,-1,-1,0],[9E+09,9E+09,9E+09,9E+09,9E+09,9E+09]];
CONST robtarget LHP_385:=[[1496.13,395.81,-167.92],[0.501832,0.0142997,0.0357903,-0.864106],[-1,-1,-1,0],[9E+09,9E+09,9E+09,9E+09,9E+09,9E+09]];
CONST robtarget LHP_390:=[[1515.01,305.29,-41.45],[0.500229,-6.95049E-05,2.93455E-05,-0.865893],[-1,-1,-1,0],[9E+09,9E+09,9E+09,9E+09,9E+09,9E+09]];
CONST robtarget LHP_395:=[[1371.85706,156.694901,-47.4344292],[0.4850808,-0.004593692,-0.00611278,-0.8744359],[-1,0,-1,0],[9E9,9E9,9E9,9E9,9E9,9E9]];
CONST robtarget LHP_400:=[[1371.81006,156.684998,-41.7470016],[0.48507392,-0.004586132,-0.006106427,-0.8744398],[-1,0,-1,0],[9E9,9E9,9E9,9E9,9E9,9E9]];
CONST robtarget LHP_405:=[[1492.72,315.84,-138.22],[0.571745,-0.00395765,-0.00657566,-0.820395],[-1,0,-1,0],[9E+09,9E+09,9E+09,9E+09,9E+09,9E+09]];
CONST robtarget LHP_410:=[[1568.64,542.95,-202.94],[0.571744,-0.00395848,-0.00658119,-0.820396],[-1,0,-1,0],[9E+09,9E+09,9E+09,9E+09,9E+09,9E+09]];
CONST robtarget LHP_415:=[[1568.58,736.45,-284.14],[0.571745,-0.00397095,-0.00657964,-0.820396],[-1,0,-1,0],[9E+09,9E+09,9E+09,9E+09,9E+09,9E+09]];
CONST robtarget LHP_420:=[[1508.30,917.00,-395.22],[0.556499,0.0508994,0.0317793,-0.828678],[-1,-1,-1,0],[9E+09,9E+09,9E+09,9E+09,9E+09,9E+09]];
CONST robtarget LHP_425:=[[1495.25,987.39,-357.83],[0.551104,0.0895725,0.0518729,-0.827992],[-1,-1,-1,0],[9E+09,9E+09,9E+09,9E+09,9E+09,9E+09]];
CONST robtarget LHP_430:=[[1328.35,635.44,-278.20],[0.501405,0.0212305,0.11734,-0.856956],[-1,-1,0,0],[9E+09,9E+09,9E+09,9E+09,9E+09,9E+09]];
CONST robtarget LHP_435:=[[1126.70,526.89,-238.13],[0.384755,0.0646485,0.107006,-0.914513],[-1,-1,0,0],[9E+09,9E+09,9E+09,9E+09,9E+09,9E+09]];
CONST robtarget LHP_440:=[[1126.70,526.87,-238.14],[0.384757,0.0646487,0.107006,-0.914512],[-1,-1,0,0],[9E+09,9E+09,9E+09,9E+09,9E+09,9E+09]];
CONST robtarget LHP_445:=[[1328.35,635.43,-278.21],[0.501406,0.0212292,0.11734,-0.856956],[-1,-1,0,0],[9E+09,9E+09,9E+09,9E+09,9E+09,9E+09]];
CONST robtarget LHP_450:=[[1495.26,987.39,-357.84],[0.551103,0.0895724,0.0518701,-0.827993],[-1,-1,-1,0],[9E+09,9E+09,9E+09,9E+09,9E+09,9E+09]];
CONST robtarget LHP_455:=[[1606.25,805.30,-336.47],[0.591189,0.0705667,0.0504833,-0.801852],[-1,-1,-1,0],[9E+09,9E+09,9E+09,9E+09,9E+09,9E+09]];
CONST robtarget LHP_460:=[[1846.21,646.41,-266.45],[0.66313,0.055392,0.0578373,-0.744207],[-1,-1,-1,0],[9E+09,9E+09,9E+09,9E+09,9E+09,9E+09]];
CONST robtarget LHP_465:=[[1831.93,634.62,-78.38],[0.625946,0.00957367,0.0100376,-0.779743],[-1,-1,-1,0],[9E+09,9E+09,9E+09,9E+09,9E+09,9E+09]];
CONST robtarget LHP_470:=[[1779.47,515.75,-42.93],[0.553641,0.000124152,-3.19163E-05,-0.832756],[-1,-1,-1,0],[9E+09,9E+09,9E+09,9E+09,9E+09,9E+09]];
CONST robtarget LHP_475:=[[1581.22,548.75,-125.86],[0.508525,0.0149425,0.00198371,-0.860915],[-1,0,-1,0],[9E+09,9E+09,9E+09,9E+09,9E+09,9E+09]];
CONST robtarget LHP_480:=[[1526.71,530.36,-111.44],[0.495097,0.0157343,0.00230728,-0.868692],[-1,0,-1,0],[9E+09,9E+09,9E+09,9E+09,9E+09,9E+09]];
CONST robtarget LHP_485:=[[1496.52905,533.620972,-169.427002],[0.5015252,0.014323151,0.035049833,-0.8643141],[-1,-1,-1,0],[9E9,9E9,9E9,9E9,9E9,9E9]];
CONST robtarget LHP_490:=[[1628.88,359.00,-167.42],[0.509965,0.00587853,-0.00326077,-0.860169],[-1,0,-1,0],[9E+09,9E+09,9E+09,9E+09,9E+09,9E+09]];
CONST robtarget LHP_495:=[[1653.10,363.04,-167.43],[0.50985,0.0307676,0.0114918,-0.859636],[-1,0,-1,0],[9E+09,9E+09,9E+09,9E+09,9E+09,9E+09]];
CONST robtarget LHP_500:=[[1734.14,581.56,-229.81],[0.51369,0.0926739,0.046858,-0.851668],[-1,-1,-1,0],[9E+09,9E+09,9E+09,9E+09,9E+09,9E+09]];
CONST robtarget LHP_505:=[[1850.77,754.32,-287.10],[0.562259,0.138379,0.0973397,-0.809469],[-1,-1,-1,0],[9E+09,9E+09,9E+09,9E+09,9E+09,9E+09]];
CONST robtarget LHP_510:=[[1850.71,883.30,-361.37],[0.589549,0.148661,0.155296,-0.778598],[-1,-1,-1,0],[9E+09,9E+09,9E+09,9E+09,9E+09,9E+09]];
CONST robtarget LHP_515:=[[1850.60,911.16,-304.76],[0.610795,0.143869,0.202267,-0.751877],[-1,-1,-1,0],[9E+09,9E+09,9E+09,9E+09,9E+09,9E+09]];
CONST robtarget LHP_520:=[[1845.93,938.54,-187.19],[0.617535,0.126482,0.223985,-0.743292],[-1,-1,-1,0],[9E+09,9E+09,9E+09,9E+09,9E+09,9E+09]];
CONST robtarget LHP_525:=[[1839.91,764.25,251.37],[0.609113,0.0794277,0.135403,-0.777392],[-1,-1,-1,0],[9E+09,9E+09,9E+09,9E+09,9E+09,9E+09]];
CONST robtarget LHP_530:=[[1951.53,815.35,1215.32],[0.610126,-0.0704393,-0.00824645,-0.789124],[-1,0,-1,0],[9E+09,9E+09,9E+09,9E+09,9E+09,9E+09]];
CONST robtarget LHP_535:=[[2438.93,960.39,2235.39],[0.671457,-0.189483,-0.125804,-0.705277],[-1,0,-1,0],[9E+09,9E+09,9E+09,9E+09,9E+09,9E+09]];
!provisorische Punkte fdz?r SP-Versetzung in Zone2
CONST robtarget LHP_605:=[[1647.70,917.36,-357.05],[0.686537,0.012902,0.00966857,-0.726916],[-1,-1,-1,0],[9E+09,9E+09,9E+09,9E+09,9E+09,9E+09]];
CONST robtarget LHP_610:=[[1610.73,498.12,-174.33],[0.637115,0.00115243,-0.000308458,-0.770768],[-1,0,-1,0],[9E+09,9E+09,9E+09,9E+09,9E+09,9E+09]];
CONST robtarget LHP_620:=[[1777.10,396.39,-174.52],[0.764298,0.00344259,-0.00243544,-0.644849],[-1,0,-1,0],[9E+09,9E+09,9E+09,9E+09,9E+09,9E+09]];
CONST robtarget LHP_625:=[[1816.72,397.75,-147.92],[0.816486,0.00152322,-0.000785194,-0.577362],[-1,0,-1,0],[9E+09,9E+09,9E+09,9E+09,9E+09,9E+09]];
CONST robtarget LHP_630:=[[1816.69,397.74,-147.92],[0.816487,0.00151316,-0.000780112,-0.577362],[-1,0,-1,0],[9E+09,9E+09,9E+09,9E+09,9E+09,9E+09]];
CONST robtarget LHP_635:=[[1517.21,788.33,-328.51],[0.603967,0.0765054,0.0409354,-0.792272],[-1,-1,-1,0],[9E+09,9E+09,9E+09,9E+09,9E+09,9E+09]];
CONST robtarget LHP_600:=[[1990.20,974.03,1486.76],[0.667207,-0.21865,0.214527,-0.678974],[-1,-1,-1,0],[9E+09,9E+09,9E+09,9E+09,9E+09,9E+09]];
! ------------------------------------------------------------
  ! Unterprogramm:
  ! Stand
  ! Daimler AG - Werk Ludwigsfelde
  ! ------------------------------------------------------------
  ! ************************************************************
  ! Kommentar: Achtung
  !            automatisch generiert!!!!!!!!!!!!!!!!!!
  ! ************************************************************

! Robotername:            1606R04
! Anlagenbezeichn:        Linie 16          Stations-Nr:  1606
! Stand / Version:        04.08.2009 / 1.1
! Name Bearbeiter:        Karmann
! Applikationssteuerung:  Punktschweissen
! Baumuster:              FHL T1 R2


INIT_SW_BASE;

WKZ_1_AUFNEHMEN;

MoveJ ToolHome1,vSchnell,fine,nomtcp1;

MoveJ LHP_000,vSchnell,fine,nomtcp1\WObj:=BS_1606_1A;

Vorhub\auf;

ABL 2\ABL_WAIT;
ABL 10\ABL_SET;

!1606R04_1606R06
KOLLISION_ZONE 2\Anfrage;
!1606R04_1606R06
KOLLISION_ZONE 7\Anfrage;
!1606R04_1606R06
KOLLISION_ZONE 9\Anfrage;

MoveJ LHP_600,vSchnell,fine,nomtcp1\WObj:=BS_1606_1A;

!
! zrobic dojazd
!
WaitUntil FALSE;


MoveJ LHP_165,vSchnell,z100,nomtcp1\WObj:=BS_1606_1A;
MoveJ LHP_160,vSchnell,z1,nomtcp1\WObj:=BS_1606_1A;
MoveJ LHP_155,vSchnell,z1,nomtcp1\WObj:=BS_1606_1A;
MoveJ LHP_150,vSchnell,z1,nomtcp1\WObj:=BS_1606_1A;

SpotL G0216190478BP20\VFO:=210,vSpot,nomtcp1\WObj:=BS_1606_1A;
SpotL G0216190582BP20\VFO:=210\Vorhub_Auf,vSpot, nomtcp1\WObj:=BS_1606_1A;

MoveJ LHP_135,vSchnell,z1,nomtcp1\WObj:=BS_1606_1A;
MoveJ LHP_130,vSchnell,z100,nomtcp1\WObj:=BS_1606_1A;

SpotL G0216190492BP20\VFO:=210\Vorhub_Auf,vSpot,nomtcp1\WObj:=BS_1606_1A;

!
! zrobic dojazd
!
WaitUntil FALSE;

KOLLISION_ZONE 2\Freigabe;

MoveJ LHP_480,vSchnell,z100,nomtcp1\WObj:=BS_1606_1A;

SpotL G0216190576BP20\VFO:=210,vSpot,nomtcp1\WObj:=BS_1606_1A;
SpotL G0213198812BP20\VFO:=210\Vorhub_Auf,vSpot,nomtcp1\WObj:=BS_1606_1A;

MoveJ LHP_485,vSchnell,z100,nomtcp1\WObj:=BS_1606_1A;

!
! zrobic dojazd
!
WaitUntil FALSE;

SpotL G0213198810BP20\VFO:=210,vSpot,nomtcp1\WObj:=BS_1606_1A;
SpotL G0213198808BP20\VFO:=210,vSpot,nomtcp1\WObj:=BS_1606_1A;
SpotL G0216021266BP20\VFO:=210,vSpot,nomtcp1\WObj:=BS_1606_1A;
SpotL G0216021268BP20\VFO:=210,vSpot,nomtcp1\WObj:=BS_1606_1A;

MoveJ LHP_470,vSchnell,fine, nomtcp1\WObj:=BS_1606_1A;

SpotL G0216021270BP20\VFO:=210\Vorhub_Auf,vSpot,nomtcp1\WObj:=BS_1606_1A;

!
! zrobic dojazd
!
WaitUntil FALSE;

MoveJ LHP_625,vSchnell,z100,nomtcp1\WObj:=BS_1606_1A;

SpotL G0216021460BP20\VFO:=210\Vorhub_Auf, vSpot, nomtcp1\WObj:=BS_1606_1A;

MoveJ LHP_630, vSchnell, z100, nomtcp1\WObj:=BS_1606_1A;

!
! zrobic dojazd
!
WaitUntil FALSE;

MoveJ LHP_025,vSchnell,z100,nomtcp1\WObj:=BS_1606_1A;
MoveJ LHP_030,vSchnell,z100,nomtcp1\WObj:=BS_1606_1A;
MoveJ LHP_035,vSchnell,z100,nomtcp1\WObj:=BS_1606_1A;

SpotL G0216021458BP20\VFO:=210,vSpot,nomtcp1\WObj:=BS_1606_1A;
SpotL G0216021456BP20\VFO:=210\Vorhub_Auf,vSpot,nomtcp1\WObj:=BS_1606_1A;

MoveJ LHP_040,vSchnell,z100,nomtcp1\WObj:=BS_1606_1A;

!
! zrobic dojazd
!
waituntil FALSE;

MoveJ LHP_465,vSchnell,z100,nomtcp1\WObj:=BS_1606_1A;
MoveJ LHP_460,vSchnell,z100,nomtcp1\WObj:=BS_1606_1A;
MoveJ LHP_455,vSchnell,z100,nomtcp1\WObj:=BS_1606_1A;
MoveJ LHP_450,vSchnell,z100,nomtcp1\WObj:=BS_1606_1A;

SpotL G0216021272BP20\VFO:=210,vSpot,nomtcp1\WObj:=BS_1606_1A;
SpotL G0216190440BP20\VFO:=210,vSpot,nomtcp1\WObj:=BS_1606_1A;
SpotL G0216190438BP20\VFO:=210,vSpot,nomtcp1\WObj:=BS_1606_1A;
SpotL G0216190436BP20\VFO:=210\Vorhub_Auf,vSpot,nomtcp1\WObj:=BS_1606_1A;

!
! zrobic dojazd
!
WaitUntil FALSE;

MoveJ LHP_445,vSchnell,z100,nomtcp1\WObj:=BS_1606_1A;

SpotL G0216190434BP20\VFO:=210,vSpot,nomtcp1\WObj:=BS_1606_1A;
SpotL G0216190432BP20\VFO:=210,vSpot,nomtcp1\WObj:=BS_1606_1A;
SpotL G0216190430BP20\VFO:=210,vSpot,nomtcp1\WObj:=BS_1606_1A;
SpotL G0216190428BP20\VFO:=210\Vorhub_Auf,vSpot,nomtcp1\WObj:=BS_1606_1A;

!
! zrobic dojazd
!
WaitUntil FALSE;

MoveJ LHP_230,vSchnell,z100,nomtcp1\WObj:=BS_1606_1A;

SpotL G0216190446BP20\VFO:=210\Vorhub_Auf,vSpot,nomtcp1\WObj:=BS_1606_1A;

KOLLISION_ZONE 1\Anfrage;
KOLLISION_ZONE 6\Anfrage;

MoveJ LHP_235,vSchnell,z100,nomtcp1\WObj:=BS_1606_1A;
MoveJ LHP_610,vSchnell,fine,nomtcp1\WObj:=BS_1606_1A;
MoveJ LHP_620,vSchnell,z100,nomtcp1\WObj:=BS_1606_1A;
MoveJ LHP_635,vSchnell,z100,nomtcp1\WObj:=BS_1606_1A;

!
! zrobic dojazd
!
WaitUntil FALSE;

MoveJ LHP_170,vSchnell,z100,nomtcp1\WObj:=BS_1606_1A;
MoveJ LHP_175,vSchnell,z100,nomtcp1\WObj:=BS_1606_1A;
MoveJ LHP_180,vSchnell,z100,nomtcp1\WObj:=BS_1606_1A;
MoveJ LHP_250,vSchnell,fine,nomtcp1\WObj:=BS_1606_1A;
MoveJ LHP_255,vSchnell,z100,nomtcp1\WObj:=BS_1606_1A;
MoveJ LHP_260,vSchnell,z100,nomtcp1\WObj:=BS_1606_1A;
MoveJ LHP_265,vSchnell,z100,nomtcp1\WObj:=BS_1606_1A;
MoveJ LHP_270,vSchnell,z100,nomtcp1\WObj:=BS_1606_1A;
MoveJ LHP_275,vSchnell,z100,nomtcp1\WObj:=BS_1606_1A;
MoveJ LHP_280,vSchnell,z100,nomtcp1\WObj:=BS_1606_1A;
MoveL LHP_285,vSchnell,z5,nomtcp1\WObj:=BS_1606_1A;
MoveL LHP_290,vSchnell,z5,nomtcp1\WObj:=BS_1606_1A;
MoveL LHP_295,vSchnell,z5,nomtcp1\WObj:=BS_1606_1A;
MoveL LHP_300,vSchnell,z5,nomtcp1\WObj:=BS_1606_1A;
MoveL LHP_305,vSchnell,z5,nomtcp1\WObj:=BS_1606_1A;

SpotL G0216190480BP20\VFO:=210\Vorhub_Auf,vSpot,nomtcp1\WObj:=BS_1606_1A;

MoveL LHP_310,vSchnell,z5,nomtcp1\WObj:=BS_1606_1A;
MoveL LHP_315,vSchnell,z5,nomtcp1\WObj:=BS_1606_1A;
MoveL LHP_320,vSchnell,z5,nomtcp1\WObj:=BS_1606_1A;
MoveL LHP_325,vSchnell,z5,nomtcp1\WObj:=BS_1606_1A;
MoveL LHP_330,vSchnell,z5,nomtcp1\WObj:=BS_1606_1A;
MoveL LHP_335,vSchnell,z5,nomtcp1\WObj:=BS_1606_1A;
MoveL LHP_340,vSchnell,z5,nomtcp1\WObj:=BS_1606_1A;

SpotL G0216022394BP20\VFO:=210\Vorhub_Auf,vSpot,nomtcp1\WObj:=BS_1606_1A;

MoveJ LHP_345,vSchnell,fine,nomtcp1\WObj:=BS_1606_1A;
MoveJ LHP_350,vSchnell,z100,nomtcp1\WObj:=BS_1606_1A;

SpotL G0216022386BP20\VFO:=210,vSpot,nomtcp1\WObj:=BS_1606_1A;

KOLLISION_ZONE 6\Freigabe;

SpotL G0216047033BP20\VFO:=210,vSpot,nomtcp1\WObj:=BS_1606_1A;
SpotL G0216047032BP20\VFO:=210\Vorhub_Auf,vSpot,nomtcp1\WObj:=BS_1606_1A;

MoveJ LHP_355,vSchnell,z100,nomtcp1\WObj:=BS_1606_1A;
MoveJ LHP_360,vSchnell,z100,nomtcp1\WObj:=BS_1606_1A;
MoveJ LHP_365,vSchnell,z100,nomtcp1\WObj:=BS_1606_1A;
MoveJ LHP_370,vSchnell,z100,nomtcp1\WObj:=BS_1606_1A;

!
! zrobic dojazd
!
WaitUntil FALSE;

MoveJ LHP_420,vSchnell,z100,nomtcp1\WObj:=BS_1606_1A;
MoveJ LHP_425,vSchnell,z100,nomtcp1\WObj:=BS_1606_1A;
MoveJ LHP_430,vSchnell,z100,nomtcp1\WObj:=BS_1606_1A;
MoveJ LHP_435,vSchnell,z100,nomtcp1\WObj:=BS_1606_1A;

SpotL G0216047028BP20\VFO:=210,vSpot,nomtcp1\WObj:=BS_1606_1A;
SpotL G0216047029BP20\VFO:=210,vSpot,nomtcp1\WObj:=BS_1606_1A;
SpotL G0216022368BP20\VFO:=210,vSpot,nomtcp1\WObj:=BS_1606_1A;
SpotL G0216022370BP20\VFO:=210\Vorhub_Auf,vSpot,nomtcp1\WObj:=BS_1606_1A;

MoveJ LHP_440,vSchnell,z100,nomtcp1\WObj:=BS_1606_1A;
MoveJ LHP_475,vSchnell,z100,nomtcp1\WObj:=BS_1606_1A;

!
! zrobic dojazd
!
WaitUntil FALSE;

SpotL G0216190516BP20\VFO:=210,vSpot,nomtcp1\WObj:=BS_1606_1A;

KOLLISION_ZONE 1\Freigabe;
KOLLISION_ZONE 7\Freigabe;
KOLLISION_ZONE 8\Anfrage;

MoveJ LHP_045,vSchnell,z100,nomtcp1\WObj:=BS_1606_1A;

SpotL G0216190518BP20\VFO:=210,vSpot,nomtcp1\WObj:=BS_1606_1A;
SpotL G0216190520BP20\VFO:=210,vSpot,nomtcp1\WObj:=BS_1606_1A;

MoveJ LHP_050,vSchnell,z100,nomtcp1\WObj:=BS_1606_1A;

SpotL G0216190522BP20\VFO:=210,vSpot,nomtcp1\WObj:=BS_1606_1A;
SpotL G0216190524BP20\VFO:=210,vSpot,nomtcp1\WObj:=BS_1606_1A;

!1606R04_1606R03
KOLLISION_ZONE 4\Anfrage;

SpotL G0216190526BP20\VFO:=210,vSpot,nomtcp1\WObj:=BS_1606_1A;
SpotL G0216190528BP20\VFO:=210\Vorhub_Auf, vSpot, nomtcp1\WObj:=BS_1606_1A;

MoveJ LHP_055,vSchnell,z100,nomtcp1\WObj:=BS_1606_1A;
MoveJ LHP_060,vSchnell,z100,nomtcp1\WObj:=BS_1606_1A;
MoveJ LHP_065,vSchnell,z100,nomtcp1\WObj:=BS_1606_1A;
MoveJ LHP_070,vSchnell,z100,nomtcp1\WObj:=BS_1606_1A;
MoveJ LHP_075,vSchnell,z100,nomtcp1\WObj:=BS_1606_1A;
MoveJ LHP_080,vSchnell,z100,nomtcp1\WObj:=BS_1606_1A;

SpotL G0216190508BP20\VFO:=210,vSpot,nomtcp1\WObj:=BS_1606_1A;

MoveJ LHP_085,vSchnell,z100,nomtcp1\WObj:=BS_1606_1A;
MoveJ LHP_090,vSchnell,z100,nomtcp1\WObj:=BS_1606_1A;

SpotL G0216190500BP20\VFO:=210\Vorhub_Auf,vSpot,nomtcp1\WObj:=BS_1606_1A;

MoveJ LHP_405,vSchnell,z100,nomtcp1\WObj:=BS_1606_1A;
MoveJ LHP_410,vSchnell,z100,nomtcp1\WObj:=BS_1606_1A;

SpotL G0216190506BP20\VFO:=210\Vorhub_Auf,vSpot,nomtcp1\WObj:=BS_1606_1A;

!
! zrobic dojazd
!
WaitUntil FALSE;

MoveJ LHP_380,vSchnell,z100,nomtcp1\WObj:=BS_1606_1A;
MoveJ LHP_385,vSchnell,z100,nomtcp1\WObj:=BS_1606_1A;
MoveJ LHP_390,vSchnell,fine,nomtcp1\WObj:=BS_1606_1A;

!1606R04_1606R06
KOLLISION_ZONE 7\Freigabe;

SpotL G0216190498BP20\VFO:=210\Vorhub_Auf,vSpot,nomtcp1\WObj:=BS_1606_1A;

MoveJ LHP_395,vSchnell,z100,nomtcp1\WObj:=BS_1606_1A;

SpotL G0216190488BP20\VFO:=210\Vorhub_Auf,vSpot,nomtcp1\WObj:=BS_1606_1A;

MoveJ LHP_400,vSchnell,z100,nomtcp1\WObj:=BS_1606_1A;

SpotL G0216190496BP20\VFO:=210,vSpot,nomtcp1\WObj:=BS_1606_1A;
SpotL G0216190494BP20\VFO:=210\Vorhub_Auf,vSpot,nomtcp1\WObj:=BS_1606_1A;

!
! zrobic dojazd
!
WaitUntil FALSE;

SpotL G0216190502BP20\VFO:=210\Vorhub_Auf,vSpot,nomtcp1\WObj:=BS_1606_1A;

KOLLISION_ZONE 8\Freigabe;

MoveJ LHP_215,vSchnell,z100,nomtcp1\WObj:=BS_1606_1A;
MoveJ LHP_220,vSchnell,z100,nomtcp1\WObj:=BS_1606_1A;

SpotL G0213198814BP20\VFO:=210\Vorhub_Auf,vSpot,nomtcp1\WObj:=BS_1606_1A;

MoveJ LHP_225,vSchnell,z100,nomtcp1\WObj:=BS_1606_1A;

!
! zrobic dojazd
!
WaitUntil FALSE;

MoveJ LHP_515,vSchnell,z5,nomtcp1\WObj:=BS_1606_1A;
MoveJ LHP_510,vSchnell,z5,nomtcp1\WObj:=BS_1606_1A;
MoveJ LHP_505,vSchnell,z5,nomtcp1\WObj:=BS_1606_1A;
MoveJ LHP_500,vSchnell,z10,nomtcp1\WObj:=BS_1606_1A;
MoveJ LHP_490,vSchnell,z100,nomtcp1\WObj:=BS_1606_1A;

SpotL G0213198816BP20\VFO:=210,vSpot,nomtcp1\WObj:=BS_1606_1A;
SpotL G0213198818BP20\VFO:=210\Vorhub_Auf,vSpot,nomtcp1\WObj:=BS_1606_1A;

MoveJ LHP_495,vSchnell,z100,nomtcp1\WObj:=BS_1606_1A;

!
! zrobic dojazd
!
waituntil FALSE;

MoveJ LHP_205,vSchnell,z100,nomtcp1\WObj:=BS_1606_1A;

SpotL G0216021464BP20\VFO:=210,vSpot,nomtcp1\WObj:=BS_1606_1A;
SpotL G0216021462BP20\VFO:=210\Vorhub_Auf,vSpot,nomtcp1\WObj:=BS_1606_1A;

!
! zrobic powrot do home
!
WaitUntil FALSE;

MoveJ LHP_520,vSchnell,z5,nomtcp1\WObj:=BS_1606_1A;
MoveJ LHP_525,vSchnell,z5,nomtcp1\WObj:=BS_1606_1A;
MoveJ LHP_530,vSchnell,fine,nomtcp1\WObj:=BS_1606_1A;

!1606R04_1606R06
KOLLISION_ZONE 1\Freigabe;

MoveJ LHP_535, vSchnell, z100, nomtcp1\WObj:=BS_1606_1A;

MoveJ ToolHome1,vSchnell,fine,nomtcp1;

ABL 254\ABL_WAIT;
ABL 255\ABL_SET;

!1606R04_1606R06
KOLLISION_ZONE 9\Freigabe;

ENDPROC





PROC swp_225300_0_st1606_1()

CONST robtarget LHP_000:=[[2573.53101,1238.19995,2660.84204],[0.56645757,-0.58473384,0.19941168,-0.54538715],[-1,-1,-1,4],[9E9,9E9,9E9,9E9,9E9,9E9]];
CONST robtarget LHP_005:=[[1933.57397,1076.34998,919.023987],[0.6739808,-0.04561597,0.22679393,-0.70159364],[-1,-1,-1,0],[9E9,9E9,9E9,9E9,9E9,9E9]];
CONST robtarget LHP_010:=[[1910.90503,994.687988,216.904999],[0.7042605,0.08468377,0.09847328,-0.6979605],[-1,-1,-1,0],[9E9,9E9,9E9,9E9,9E9,9E9]];
CONST robtarget LHP_015:=[[1910.89099,994.690002,-385.321991],[0.683501,0.087539785,0.09595496,-0.71830064],[-1,-1,-1,0],[9E9,9E9,9E9,9E9,9E9,9E9]];
CONST robtarget LHP_020:=[[1910.92,803.63,-358.65],[0.683496,0.087554,0.0959515,-0.718305],[-1,-1,-1,0],[9E+09,9E+09,9E+09,9E+09,9E+09,9E+09]];
CONST robtarget LHP_025:=[[1910.97,741.50,-281.66],[0.683494,0.0875455,0.0959486,-0.718307],[-1,-1,-1,0],[9E+09,9E+09,9E+09,9E+09,9E+09,9E+09]];
CONST robtarget LHP_030:=[[1910.91,559.83,-213.69],[0.686476,0.0613746,0.0695917,-0.721208],[-1,-1,-1,0],[9E+09,9E+09,9E+09,9E+09,9E+09,9E+09]];
CONST robtarget LHP_035:=[[1929.33,361.88,-170.13],[0.702471,0.0120548,-0.002609,-0.711605],[-1,0,-1,0],[9E+09,9E+09,9E+09,9E+09,9E+09,9E+09]];
CONST robtarget LHP_040:=[[2007.526,383.55899,-50.7519989],[0.75072795,0.000611088,0.00040383,-0.6606111],[-1,-1,-1,0],[9E9,9E9,9E9,9E9,9E9,9E9]];
CONST robtarget LHP_045:=[[1993.04797,313.046997,-31.7070007],[0.7336252,0.009941696,-0.001285905,-0.67948043],[-1,0,-1,0],[9E9,9E9,9E9,9E9,9E9,9E9]];
CONST robtarget LHP_050:=[[2002.59399,189.292999,-35.1940002],[0.73792726,0.009937888,-0.0012356,-0.67480594],[-1,0,-1,0],[9E9,9E9,9E9,9E9,9E9,9E9]];
CONST robtarget LHP_055:=[[1987.44,-5.82,-69.73],[0.747483,0.000551369,0.000433351,-0.664281],[-1,-1,-1,0],[9E+09,9E+09,9E+09,9E+09,9E+09,9E+09]];
CONST robtarget LHP_060:=[[1929.34,361.89,-170.15],[0.70247,0.0120598,-0.00260928,-0.711607],[-1,0,-1,0],[9E+09,9E+09,9E+09,9E+09,9E+09,9E+09]];
CONST robtarget LHP_065:=[[1910.91,559.85,-213.71],[0.686472,0.0613779,0.0695915,-0.721211],[-1,-1,-1,0],[9E+09,9E+09,9E+09,9E+09,9E+09,9E+09]];
CONST robtarget LHP_070:=[[1769.54,626.69,-228.36],[0.648406,0.063605,0.0595836,-0.756289],[-1,-1,-1,0],[9E+09,9E+09,9E+09,9E+09,9E+09,9E+09]];
CONST robtarget LHP_075:=[[1629.23,373.82,-175.88],[0.60566,0.011527,-0.00436593,-0.795628],[-1,0,-1,0],[9E+09,9E+09,9E+09,9E+09,9E+09,9E+09]];
CONST robtarget LHP_080:=[[1643.37,44.45,-93.67],[0.638426,0.0118697,-0.00343011,-0.769584],[-1,0,-1,0],[9E+09,9E+09,9E+09,9E+09,9E+09,9E+09]];
CONST robtarget LHP_085:=[[1645.79,51.65,-47.78],[0.621544,0.019299,-0.00963586,-0.783082],[-1,0,-1,0],[9E+09,9E+09,9E+09,9E+09,9E+09,9E+09]];
CONST robtarget LHP_090:=[[1652.62,133.53,-52.42],[0.605581,0.0130855,-0.00581803,-0.795655],[-1,0,-1,0],[9E+09,9E+09,9E+09,9E+09,9E+09,9E+09]];
CONST robtarget LHP_095:=[[1617.10803,350.912994,-180.268005],[0.56401443,0.037766688,0.053717423,-0.8231499],[-1,-1,-1,0],[9E9,9E9,9E9,9E9,9E9,9E9]];
CONST robtarget LHP_100:=[[1517.84,635.47,-254.71],[0.565141,-0.00404407,-0.00655324,-0.824958],[-1,0,-1,0],[9E+09,9E+09,9E+09,9E+09,9E+09,9E+09]];
CONST robtarget LHP_105:=[[1647.70,917.36,-357.05],[0.686537,0.012902,0.00966857,-0.726916],[-1,-1,-1,0],[9E+09,9E+09,9E+09,9E+09,9E+09,9E+09]];
CONST robtarget LHP_110:=[[1402.01,954.02,-347.18],[0.618002,-0.00350893,0.00682793,-0.786139],[-1,-1,-1,0],[9E+09,9E+09,9E+09,9E+09,9E+09,9E+09]];
CONST robtarget LHP_115:=[[1380.13,800.38,-342.28],[0.663576,-0.00391562,0.00660285,-0.74807],[-1,-1,-1,0],[9E+09,9E+09,9E+09,9E+09,9E+09,9E+09]];
CONST robtarget LHP_120:=[[1355.05,688.92,-230.68],[0.643458,-0.00406434,0.0069742,-0.765439],[-1,-1,-1,0],[9E+09,9E+09,9E+09,9E+09,9E+09,9E+09]];
CONST robtarget LHP_125:=[[1338.98,616.80,-217.15],[0.641931,-0.00377363,0.00673657,-0.766724],[-1,-1,-1,0],[9E+09,9E+09,9E+09,9E+09,9E+09,9E+09]];
CONST robtarget LHP_130:=[[1328.82,551.60,-198.45],[0.643236,-0.00380631,0.00669098,-0.765629],[-1,-1,-1,0],[9E+09,9E+09,9E+09,9E+09,9E+09,9E+09]];
CONST robtarget LHP_135:=[[1301.19,432.03,-200.08],[0.630965,0.0270779,0.0228783,-0.775001],[-1,-1,-1,0],[9E+09,9E+09,9E+09,9E+09,9E+09,9E+09]];
CONST robtarget LHP_140:=[[1315.22,418.75,-159.95],[0.640955,0.052567,0.0459758,-0.764395],[-1,-1,-1,0],[9E+09,9E+09,9E+09,9E+09,9E+09,9E+09]];
CONST robtarget LHP_145:=[[1314.89,402.01,-58.59],[0.643636,0.0406528,0.0359674,-0.763405],[-1,-1,-1,0],[9E+09,9E+09,9E+09,9E+09,9E+09,9E+09]];
CONST robtarget LHP_150:=[[1314.89,402.00,-58.59],[0.64363700,0.04065100,0.0359677,-0.7634040],[-1,-1,-1,0],[9E+09,9E+09,9E+09,9E+09,9E+09,9E+09]];
CONST robtarget LHP_155:=[[1315.25,418.75,-159.98],[0.640959,0.05257270,0.04597540,-0.7643910],[-1,-1,-1,0],[9E+09,9E+09,9E+09,9E+09,9E+09,9E+09]];
CONST robtarget LHP_160:=[[1301.20,432.03,-200.09],[0.630966,0.0270787,0.0228773,-0.775],[-1,-1,-1,0],[9E+09,9E+09,9E+09,9E+09,9E+09,9E+09]];
CONST robtarget LHP_165:=[[1328.84,551.60,-198.48],[0.643767,-0.00379566,0.00669219,-0.765183],[-1,-1,-1,0],[9E+09,9E+09,9E+09,9E+09,9E+09,9E+09]];
CONST robtarget LHP_170:=[[1356.81,663.69,-214.66],[0.64609,-0.00377796,0.00670482,-0.7632220],[-1,-1,-1,0],[9E+09,9E+09,9E+09,9E+09,9E+09,9E+09]];
CONST robtarget LHP_175:=[[1392.09,854.35,-337.39],[0.646086,-0.00378978,0.00670626,-0.763226],[-1,-1,-1,0],[9E+09,9E+09,9E+09,9E+09,9E+09,9E+09]];
CONST robtarget LHP_180:=[[1392.10,915.32,-339.98],[0.646085,-0.00379686,0.00670629,-0.763227],[-1,-1,-1,0],[9E+09,9E+09,9E+09,9E+09,9E+09,9E+09]];
CONST robtarget LHP_185:=[[1392.13,915.34,-336.92],[0.646086,-0.00378783,0.00670572,-0.763226],[-1,-1,-1,0],[9E+09,9E+09,9E+09,9E+09,9E+09,9E+09]];
CONST robtarget LHP_190:=[[1777.10,396.39,-174.51],[0.778298,0.00338922,-0.00251072,-0.62788],[-1,0,-1,0],[9E+09,9E+09,9E+09,9E+09,9E+09,9E+09]];
CONST robtarget LHP_195:=[[1816.72,397.75,-147.92],[0.816486,0.00152322,-0.000785194,-0.577362],[-1,0,-1,0],[9E+09,9E+09,9E+09,9E+09,9E+09,9E+09]];
CONST robtarget LHP_200:=[[1816.69,397.74,-147.92],[0.816487,0.00151316,-0.000780112,-0.577362],[-1,0,-1,0],[9E+09,9E+09,9E+09,9E+09,9E+09,9E+09]];
CONST robtarget LHP_205:=[[1684.99,383.29,-52.10],[0.598242,-0.000451381,-0.0146486,-0.801182],[-1,0,-1,0],[9E+09,9E+09,9E+09,9E+09,9E+09,9E+09]];
CONST robtarget LHP_210:=[[1517.37,845.68,-347.51],[0.603966,0.0765094,0.0409368,-0.792272],[-1,-1,-1,0],[9E+09,9E+09,9E+09,9E+09,9E+09,9E+09]];
CONST robtarget LHP_215:=[[1614.81,303.29,-114.97],[0.595541,4.37463E-06,7.52158E-05,-0.803325],[-1,-1,-1,0],[9E+09,9E+09,9E+09,9E+09,9E+09,9E+09]];
CONST robtarget LHP_220:=[[1496.10,381.00,-140.90],[0.501832,0.0142883,0.0357857,-0.864106],[-1,-1,-1,0],[9E+09,9E+09,9E+09,9E+09,9E+09,9E+09]];
CONST robtarget LHP_225:=[[1496.16,381.04,-179.37],[0.501836,0.0143261,0.0358019,-0.864103],[-1,-1,-1,0],[9E+09,9E+09,9E+09,9E+09,9E+09,9E+09]];
CONST robtarget LHP_230:=[[1517.37,556.59,-186.35],[0.545787,0.0365786,0.0545327,-0.835347],[-1,-1,-1,0],[9E+09,9E+09,9E+09,9E+09,9E+09,9E+09]];
CONST robtarget LHP_235:=[[1529.66,619.50,-150.47],[0.565262,-0.000227126,0.000165536,-0.824912],[-1,-1,-1,0],[9E+09,9E+09,9E+09,9E+09,9E+09,9E+09]];
CONST robtarget LHP_240:=[[1558.44,796.09,-349.49],[0.583985,0.0684408,0.0319346,-0.808244],[-1,-1,-1,0],[9E+09,9E+09,9E+09,9E+09,9E+09,9E+09]];
CONST robtarget LHP_245:=[[1477.93,985.71,-357.82],[0.551096,0.0897034,0.0519627,-0.827978],[-1,-1,-1,0],[9E+09,9E+09,9E+09,9E+09,9E+09,9E+09]];
CONST robtarget LHP_250:=[[807.86,896.51,-348.98],[0.475989,-0.019585,0.0486327,-0.877887],[-1,-1,-1,0],[9E+09,9E+09,9E+09,9E+09,9E+09,9E+09]];
CONST robtarget LHP_255:=[[807.84,813.89,-348.98],[0.47599,-0.0195894,0.0486332,-0.877887],[-1,-1,-1,0],[9E+09,9E+09,9E+09,9E+09,9E+09,9E+09]];
CONST robtarget LHP_260:=[[798.625,757.187988,-251.093002],[0.47488588,-0.019798715,0.048936285,-0.8784627],[-1,-1,-1,0],[9E9,9E9,9E9,9E9,9E9,9E9]];
CONST robtarget LHP_265:=[[687.672974,377.386993,-182.552002],[0.5034063,-0.04137853,0.03811411,-0.8622165],[-1,-1,-1,0],[9E9,9E9,9E9,9E9,9E9,9E9]];
CONST robtarget LHP_270:=[[796.06,403.61,2.12],[0.54967,-0.0809587,0.0198978,-0.831212],[-1,-1,-1,0],[9E+09,9E+09,9E+09,9E+09,9E+09,9E+09]];
CONST robtarget LHP_275:=[[951.56,404.05,-36.64],[0.666081,-0.0483269,0.018538,-0.744081],[-1,-1,-1,0],[9E+09,9E+09,9E+09,9E+09,9E+09,9E+09]];
CONST robtarget LHP_280:=[[1053.17,384.08,-147.35],[0.741703,0.0276666,0.0554714,-0.667858],[-1,-1,-1,0],[9E+09,9E+09,9E+09,9E+09,9E+09,9E+09]];
CONST robtarget LHP_285:=[[1117.00,437.68,-186.63],[0.764604,0.0628167,0.0737039,-0.637183],[-1,-1,-1,0],[9E+09,9E+09,9E+09,9E+09,9E+09,9E+09]];
CONST robtarget LHP_290:=[[1206.43,437.70,-186.66],[0.808318,0.0679399,0.0690137,-0.580726],[-1,-1,-1,0],[9E+09,9E+09,9E+09,9E+09,9E+09,9E+09]];
CONST robtarget LHP_295:=[[1254.01,306.17,-147.47],[0.819239,0.0692406,0.0677067,-0.565215],[-1,-1,-1,0],[9E+09,9E+09,9E+09,9E+09,9E+09,9E+09]];
CONST robtarget LHP_300:=[[1294.76,251.64,-118.31],[0.839473,0.0657832,0.0563212,-0.536456],[-1,-1,-1,0],[9E+09,9E+09,9E+09,9E+09,9E+09,9E+09]];
CONST robtarget LHP_305:=[[1302.68,268.91,-77.08],[0.850295,0.0194976,0.0312356,-0.525017],[-1,-1,-1,0],[9E+09,9E+09,9E+09,9E+09,9E+09,9E+09]];
CONST robtarget LHP_310:=[[1302.67,268.92,-77.09],[0.850295,0.0194964,0.0312402,-0.525016],[-1,-1,-1,0],[9E+09,9E+09,9E+09,9E+09,9E+09,9E+09]];
CONST robtarget LHP_315:=[[1294.76,251.64,-118.31],[0.839473,0.0657839,0.0563209,-0.536456],[-1,-1,-1,0],[9E+09,9E+09,9E+09,9E+09,9E+09,9E+09]];
CONST robtarget LHP_320:=[[1254.01,306.17,-147.47],[0.819239,0.0692405,0.0677067,-0.565215],[-1,-1,-1,0],[9E+09,9E+09,9E+09,9E+09,9E+09,9E+09]];
CONST robtarget LHP_325:=[[1206.43,437.70,-186.66],[0.808318,0.0679399,0.0690137,-0.580726],[-1,-1,-1,0],[9E+09,9E+09,9E+09,9E+09,9E+09,9E+09]];
CONST robtarget LHP_330:=[[1117.00,437.68,-186.63],[0.764604,0.0628167,0.0737039,-0.637183],[-1,-1,-1,0],[9E+09,9E+09,9E+09,9E+09,9E+09,9E+09]];
CONST robtarget LHP_335:=[[1116.98,404.12,-155.12],[0.767929,0.0632076,0.0733697,-0.633172],[-1,-1,-1,0],[9E+09,9E+09,9E+09,9E+09,9E+09,9E+09]];
CONST robtarget LHP_340:=[[1116.98,404.12,-77.86],[0.763388,0.0288222,0.0341692,-0.644392],[-1,-1,-1,0],[9E+09,9E+09,9E+09,9E+09,9E+09,9E+09]];
CONST robtarget LHP_345:=[[951.56,404.05,-36.63],[0.666079,-0.0483271,0.018537,-0.744083],[-1,-1,-1,0],[9E+09,9E+09,9E+09,9E+09,9E+09,9E+09]];
CONST robtarget LHP_350:=[[863.42,413.34,0.81],[0.590286,-0.0726155,0.0279581,-0.803435],[-1,-1,-1,0],[9E+09,9E+09,9E+09,9E+09,9E+09,9E+09]];
CONST robtarget LHP_355:=[[687.66803,377.371002,-182.531006],[0.5034058,-0.04138605,0.0381097,-0.8622166],[-1,-1,-1,0],[9E9,9E9,9E9,9E9,9E9,9E9]];
CONST robtarget LHP_360:=[[798.580994,757.198975,-251.070007],[0.47486982,-0.019813199,0.04892835,-0.8784715],[-1,-1,-1,0],[9E9,9E9,9E9,9E9,9E9,9E9]];
CONST robtarget LHP_365:=[[961.40,981.11,-456.97],[0.440335,0.0935079,0.0750373,-0.889792],[-1,-1,-1,0],[9E+09,9E+09,9E+09,9E+09,9E+09,9E+09]];
CONST robtarget LHP_370:=[[1477.90,985.72,-357.83],[0.558631,0.0901634,0.0511329,-0.822914],[-1,-1,-1,0],[9E+09,9E+09,9E+09,9E+09,9E+09,9E+09]];
CONST robtarget LHP_375:=[[1538.22,786.86,-339.64],[0.544053,0.0691445,0.0535195,-0.834482],[-1,-1,-1,0],[9E+09,9E+09,9E+09,9E+09,9E+09,9E+09]];
CONST robtarget LHP_380:=[[1502.92,670.32,-266.02],[0.529086,0.0479959,0.0506422,-0.845695],[-1,-1,-1,0],[9E+09,9E+09,9E+09,9E+09,9E+09,9E+09]];
CONST robtarget LHP_385:=[[1496.13,395.81,-167.92],[0.501832,0.0142997,0.0357903,-0.864106],[-1,-1,-1,0],[9E+09,9E+09,9E+09,9E+09,9E+09,9E+09]];
CONST robtarget LHP_390:=[[1515.01,305.29,-41.45],[0.500229,-6.95049E-05,2.93455E-05,-0.865893],[-1,-1,-1,0],[9E+09,9E+09,9E+09,9E+09,9E+09,9E+09]];
CONST robtarget LHP_395:=[[1371.85706,156.694901,-47.4344292],[0.4850808,-0.004593692,-0.00611278,-0.8744359],[-1,0,-1,0],[9E9,9E9,9E9,9E9,9E9,9E9]];
CONST robtarget LHP_400:=[[1371.81006,156.684998,-41.7470016],[0.48507392,-0.004586132,-0.006106427,-0.8744398],[-1,0,-1,0],[9E9,9E9,9E9,9E9,9E9,9E9]];
CONST robtarget LHP_405:=[[1492.72,315.84,-138.22],[0.571745,-0.00395765,-0.00657566,-0.820395],[-1,0,-1,0],[9E+09,9E+09,9E+09,9E+09,9E+09,9E+09]];
CONST robtarget LHP_410:=[[1568.64,542.95,-202.94],[0.571744,-0.00395848,-0.00658119,-0.820396],[-1,0,-1,0],[9E+09,9E+09,9E+09,9E+09,9E+09,9E+09]];
CONST robtarget LHP_415:=[[1568.58,736.45,-284.14],[0.571745,-0.00397095,-0.00657964,-0.820396],[-1,0,-1,0],[9E+09,9E+09,9E+09,9E+09,9E+09,9E+09]];
CONST robtarget LHP_420:=[[1508.30,917.00,-395.22],[0.556499,0.0508994,0.0317793,-0.828678],[-1,-1,-1,0],[9E+09,9E+09,9E+09,9E+09,9E+09,9E+09]];
CONST robtarget LHP_425:=[[1495.25,987.39,-357.83],[0.551104,0.0895725,0.0518729,-0.827992],[-1,-1,-1,0],[9E+09,9E+09,9E+09,9E+09,9E+09,9E+09]];
CONST robtarget LHP_430:=[[1328.35,635.44,-278.20],[0.501405,0.0212305,0.11734,-0.856956],[-1,-1,0,0],[9E+09,9E+09,9E+09,9E+09,9E+09,9E+09]];
CONST robtarget LHP_435:=[[1126.70,526.89,-238.13],[0.384755,0.0646485,0.107006,-0.914513],[-1,-1,0,0],[9E+09,9E+09,9E+09,9E+09,9E+09,9E+09]];
CONST robtarget LHP_440:=[[1126.70,526.87,-238.14],[0.384757,0.0646487,0.107006,-0.914512],[-1,-1,0,0],[9E+09,9E+09,9E+09,9E+09,9E+09,9E+09]];
CONST robtarget LHP_445:=[[1328.35,635.43,-278.21],[0.501406,0.0212292,0.11734,-0.856956],[-1,-1,0,0],[9E+09,9E+09,9E+09,9E+09,9E+09,9E+09]];
CONST robtarget LHP_450:=[[1495.26,987.39,-357.84],[0.551103,0.0895724,0.0518701,-0.827993],[-1,-1,-1,0],[9E+09,9E+09,9E+09,9E+09,9E+09,9E+09]];
CONST robtarget LHP_455:=[[1606.25,805.30,-336.47],[0.591189,0.0705667,0.0504833,-0.801852],[-1,-1,-1,0],[9E+09,9E+09,9E+09,9E+09,9E+09,9E+09]];
CONST robtarget LHP_460:=[[1846.21,646.41,-266.45],[0.66313,0.055392,0.0578373,-0.744207],[-1,-1,-1,0],[9E+09,9E+09,9E+09,9E+09,9E+09,9E+09]];
CONST robtarget LHP_465:=[[1831.93,634.62,-78.38],[0.625946,0.00957367,0.0100376,-0.779743],[-1,-1,-1,0],[9E+09,9E+09,9E+09,9E+09,9E+09,9E+09]];
CONST robtarget LHP_470:=[[1793.13,513.60,-41.97],[0.578209,9.78811E-06,-2.13769E-07,-0.815889],[-1,-1,-1,0],[9E+09,9E+09,9E+09,9E+09,9E+09,9E+09]];
CONST robtarget LHP_475:=[[1581.22,548.75,-125.86],[0.508525,0.0149425,0.00198371,-0.860915],[-1,0,-1,0],[9E+09,9E+09,9E+09,9E+09,9E+09,9E+09]];
CONST robtarget LHP_480:=[[1526.71,530.36,-111.44],[0.495097,0.0157343,0.00230728,-0.868692],[-1,0,-1,0],[9E+09,9E+09,9E+09,9E+09,9E+09,9E+09]];
CONST robtarget LHP_485:=[[1496.52905,533.620972,-169.427002],[0.5015252,0.014323151,0.035049833,-0.8643141],[-1,-1,-1,0],[9E9,9E9,9E9,9E9,9E9,9E9]];
CONST robtarget LHP_490:=[[1628.88,359.00,-167.42],[0.509965,0.00587853,-0.00326077,-0.860169],[-1,0,-1,0],[9E+09,9E+09,9E+09,9E+09,9E+09,9E+09]];
CONST robtarget LHP_495:=[[1653.10,363.04,-167.43],[0.50985,0.0307676,0.0114918,-0.859636],[-1,0,-1,0],[9E+09,9E+09,9E+09,9E+09,9E+09,9E+09]];
CONST robtarget LHP_500:=[[1734.14,581.56,-229.81],[0.51369,0.0926739,0.046858,-0.851668],[-1,-1,-1,0],[9E+09,9E+09,9E+09,9E+09,9E+09,9E+09]];
CONST robtarget LHP_505:=[[1850.77,754.32,-287.10],[0.562259,0.138379,0.0973397,-0.809469],[-1,-1,-1,0],[9E+09,9E+09,9E+09,9E+09,9E+09,9E+09]];
CONST robtarget LHP_510:=[[1850.71,883.30,-361.37],[0.589549,0.148661,0.155296,-0.778598],[-1,-1,-1,0],[9E+09,9E+09,9E+09,9E+09,9E+09,9E+09]];
CONST robtarget LHP_515:=[[1850.60,911.16,-304.76],[0.610795,0.143869,0.202267,-0.751877],[-1,-1,-1,0],[9E+09,9E+09,9E+09,9E+09,9E+09,9E+09]];
CONST robtarget LHP_520:=[[1845.93,938.54,-187.19],[0.617535,0.126482,0.223985,-0.743292],[-1,-1,-1,0],[9E+09,9E+09,9E+09,9E+09,9E+09,9E+09]];
CONST robtarget LHP_525:=[[1839.91,764.25,251.37],[0.609113,0.0794277,0.135403,-0.777392],[-1,-1,-1,0],[9E+09,9E+09,9E+09,9E+09,9E+09,9E+09]];
CONST robtarget LHP_530:=[[1951.53,815.35,1215.32],[0.610126,-0.0704393,-0.00824645,-0.789124],[-1,0,-1,0],[9E+09,9E+09,9E+09,9E+09,9E+09,9E+09]];
CONST robtarget LHP_535:=[[2438.93,960.39,2235.39],[0.671457,-0.189483,-0.125804,-0.705277],[-1,0,-1,0],[9E+09,9E+09,9E+09,9E+09,9E+09,9E+09]];
!provisorische Punkte fdz?r SP-Versetzung in Zone2
CONST robtarget LHP_605:=[[1647.70,917.36,-357.05],[0.686537,0.012902,0.00966857,-0.726916],[-1,-1,-1,0],[9E+09,9E+09,9E+09,9E+09,9E+09,9E+09]];
CONST robtarget LHP_610:=[[1620.32,602.14,-205.68],[0.637115,0.00115264,-0.000310519,-0.770768],[-1,0,-1,0],[9E+09,9E+09,9E+09,9E+09,9E+09,9E+09]];
CONST robtarget LHP_620:=[[1912.93,601.14,-205.68],[0.710988,0.0011134,-0.000423279,-0.703204],[-1,0,-1,0],[9E+09,9E+09,9E+09,9E+09,9E+09,9E+09]];
CONST robtarget LHP_625:=[[1919.94,393.08,-177.19],[0.710987,0.00110842,-0.000423915,-0.703204],[-1,0,-1,0],[9E+09,9E+09,9E+09,9E+09,9E+09,9E+09]];
CONST robtarget LHP_630:=[[1919.96,393.09,-177.22],[0.710988,0.0011168,-0.000424803,-0.703203],[-1,0,-1,0],[9E+09,9E+09,9E+09,9E+09,9E+09,9E+09]];
CONST robtarget LHP_635:=[[1912.96,653.53,-205.68],[0.710987,0.00111256,-0.000425587,-0.703204],[-1,0,-1,0],[9E+09,9E+09,9E+09,9E+09,9E+09,9E+09]];
CONST robtarget LHP_600:=[[1990.20,974.03,1486.76],[0.667207,-0.21865,0.214527,-0.678974],[-1,-1,-1,0],[9E+09,9E+09,9E+09,9E+09,9E+09,9E+09]];
! ------------------------------------------------------------
! Unterprogramm:
! Stand
! Daimler AG - Werk Ludwigsfelde
! ------------------------------------------------------------
! ************************************************************
! Kommentar: Achtung
! automatisch generiert!!!!!!!!!!!!!!!!!!
! ************************************************************

! Robotername: 1606R04
! Anlagenbezeichn: Linie 16 Stations-Nr: 1606
! Stand / Version: 04.08.2009 / 1.1
! Name Bearbeiter: Karmann
! Applikationssteuerung: Punktschweissen
! Baumuster: FHL T1 R2


INIT_SW_BASE;

WKZ_1_AUFNEHMEN;
!
MoveJ ToolHome1,vSchnell,fine,nomtcp1;
!
MoveJ LHP_000,vSchnell,fine,nomtcp1\WObj:=BS_1606_1A;
!
Vorhub\auf;
!
ABL 2\ABL_WAIT;
!
ABL 10\ABL_SET;

!
!1606R04_1606R06
KOLLISION_ZONE 6\Anfrage;
!
!1606R04_1606R06
KOLLISION_ZONE 7\Anfrage;
!
!1606R04_1606R06
KOLLISION_ZONE 8\Anfrage;
!
MoveJ LHP_600, vSchnell, fine, nomtcp1\WObj:=BS_1606_1A;
!
!1606R04_1606R06
KOLLISION_ZONE 1\Anfrage;
!
MoveJ LHP_005,vSchnell,z100,nomtcp1\WObj:=BS_1606_1A;
MoveJ LHP_010,vSchnell,z100,nomtcp1\WObj:=BS_1606_1A;
MoveJ LHP_015,vSchnell,z100,nomtcp1\WObj:=BS_1606_1A;
MoveJ LHP_020,vSchnell,z100,nomtcp1\WObj:=BS_1606_1A;
MoveJ LHP_025,vSchnell,z100,nomtcp1\WObj:=BS_1606_1A;
MoveJ LHP_030,vSchnell,z100,nomtcp1\WObj:=BS_1606_1A;
MoveJ LHP_035, vSchnell, z100, nomtcp1\WObj:=BS_1606_1A;
!
SpotL G0216023180BP20\VFO:=210,vSpot,nomtcp1\WObj:=BS_1606_1A;
!
MoveJ LHP_040,vSchnell,z100,nomtcp1\WObj:=BS_1606_1A;
!
SpotL G0216190516BP20\VFO:=210,vSpot,nomtcp1\WObj:=BS_1606_1A;
!
MoveJ LHP_045,vSchnell,z100,nomtcp1\WObj:=BS_1606_1A;
!
SpotL G0216190518BP20\VFO:=210,vSpot,nomtcp1\WObj:=BS_1606_1A;
!
SpotL G0216190520BP20\VFO:=210,vSpot,nomtcp1\WObj:=BS_1606_1A;
!
MoveJ LHP_050,vSchnell,z100,nomtcp1\WObj:=BS_1606_1A;
!
SpotL G0216190522BP20\VFO:=210,vSpot,nomtcp1\WObj:=BS_1606_1A;
!
SpotL G0216190524BP20\VFO:=210,vSpot,nomtcp1\WObj:=BS_1606_1A;
!
!1606R04_1606R03
KOLLISION_ZONE 4\Anfrage;
!
SpotL G0216190526BP20\VFO:=210,vSpot,nomtcp1\WObj:=BS_1606_1A;
!
SpotL G0216190528BP20\VFO:=210\Vorhub_Auf, vSpot, nomtcp1\WObj:=BS_1606_1A;
!
MoveJ LHP_055,vSchnell,z100,nomtcp1\WObj:=BS_1606_1A;
MoveJ LHP_060,vSchnell,z100,nomtcp1\WObj:=BS_1606_1A;
MoveJ LHP_065,vSchnell,z100,nomtcp1\WObj:=BS_1606_1A;
MoveJ LHP_070,vSchnell,z100,nomtcp1\WObj:=BS_1606_1A;
MoveJ LHP_075,vSchnell,z100,nomtcp1\WObj:=BS_1606_1A;
MoveJ LHP_080,vSchnell,z100,nomtcp1\WObj:=BS_1606_1A;
!
SpotL G0216190508BP20\VFO:=210,vSpot,nomtcp1\WObj:=BS_1606_1A;
!
MoveJ LHP_085,vSchnell,z100,nomtcp1\WObj:=BS_1606_1A;
MoveJ LHP_090,vSchnell,z100,nomtcp1\WObj:=BS_1606_1A;
!
SpotL G0216190506BP20\VFO:=210, vSpot, nomtcp1\WObj:=BS_1606_1A;
!
!1606R04_1606R03
KOLLISION_ZONE 4\Freigabe;
!
MoveJ LHP_205,vSchnell,z100,nomtcp1\WObj:=BS_1606_1A;
!
SpotL G0216023184BP20\VFO:=210, vSpot, nomtcp1\WObj:=BS_1606_1A;
!
SpotL G0216023186BP20\VFO:=210, vSpot, nomtcp1\WObj:=BS_1606_1A;
!
SpotL G0216190502BP20\VFO:=210\Vorhub_Auf, vSpot, nomtcp1\WObj:=BS_1606_1A;
!
MoveJ LHP_215, vSchnell, z100, nomtcp1\WObj:=BS_1606_1A;
MoveJ LHP_220, vSchnell, z100, nomtcp1\WObj:=BS_1606_1A;
!
!
SpotL G0213195684BP20\VFO:=210\Vorhub_Auf, vSpot, nomtcp1\WObj:=BS_1606_1A;
!
MoveJ LHP_225, vSchnell, z100, nomtcp1\WObj:=BS_1606_1A;
MoveJ LHP_230,vSchnell,z100,nomtcp1\WObj:=BS_1606_1A;
!
SpotL G0216190446BP20\VFO:=210\Vorhub_Auf,vSpot,nomtcp1\WObj:=BS_1606_1A;
!
MoveJ LHP_235,vSchnell,z100,nomtcp1\WObj:=BS_1606_1A;
MoveJ LHP_610, vSchnell, fine, nomtcp1\WObj:=BS_1606_1A;
!
!1606R04_1606R06
KOLLISION_ZONE 2\Anfrage;
!
MoveJ LHP_620,vSchnell,z100,nomtcp1\WObj:=BS_1606_1A;
MoveJ LHP_625,vSchnell,z100,nomtcp1\WObj:=BS_1606_1A;
!
SpotL G0216023182BP20\VFO:=210\Vorhub_Auf, vSpot, nomtcp1\WObj:=BS_1606_1A;
!
MoveJ LHP_630, vSchnell, z100, nomtcp1\WObj:=BS_1606_1A;
MoveJ LHP_635, vSchnell, z100, nomtcp1\WObj:=BS_1606_1A;
MoveJ LHP_645, vSchnell, z100, nomtcp1\WObj:=BS_1606_1A;
MoveJ LHP_115,vSchnell,z100,nomtcp1\WObj:=BS_1606_1A;
MoveJ LHP_120,vSchnell,z100,nomtcp1\WObj:=BS_1606_1A;
MoveJ LHP_125,vSchnell,z100,nomtcp1\WObj:=BS_1606_1A;
!
SpotL G0216190492BP20\VFO:=220\Vorhub_Auf,vSpot,nomtcp1\WObj:=BS_1606_1A;
!
MoveJ LHP_130,vSchnell,z100,nomtcp1\WObj:=BS_1606_1A;
MoveJ LHP_135,vSchnell,z1,nomtcp1\WObj:=BS_1606_1A;
MoveL LHP_140,vSchnell,z1,nomtcp1\WObj:=BS_1606_1A;
MoveL LHP_145,vSchnell,z1,nomtcp1\WObj:=BS_1606_1A;
!
SpotL G0216190582BP20\VFO:=210, vSpot, nomtcp1\WObj:=BS_1606_1A;
!
SpotL G0216190478BP20\VFO:=210\Vorhub_Auf,vSpot,nomtcp1\WObj:=BS_1606_1A;
!
MoveJ LHP_150,vSchnell,z1,nomtcp1\WObj:=BS_1606_1A;
MoveJ LHP_155,vSchnell,z1,nomtcp1\WObj:=BS_1606_1A;
MoveJ LHP_160,vSchnell,z1,nomtcp1\WObj:=BS_1606_1A;
MoveJ LHP_165,vSchnell,z100,nomtcp1\WObj:=BS_1606_1A;
MoveJ LHP_170,vSchnell,z100,nomtcp1\WObj:=BS_1606_1A;
MoveJ LHP_175,vSchnell,z100,nomtcp1\WObj:=BS_1606_1A;
MoveJ LHP_180, vSchnell, z100, nomtcp1\WObj:=BS_1606_1A;
!
!1606R04_1606R06
KOLLISION_ZONE 2\Freigabe;
!
MoveJ LHP_250, vSchnell, fine, nomtcp1\WObj:=BS_1606_1A;
!1606R04_1606R06
KOLLISION_ZONE 5\Anfrage;
!
MoveJ LHP_255,vSchnell,z100,nomtcp1\WObj:=BS_1606_1A;
MoveJ LHP_260,vSchnell,z100,nomtcp1\WObj:=BS_1606_1A;
MoveJ LHP_265,vSchnell,z100,nomtcp1\WObj:=BS_1606_1A;
MoveJ LHP_270,vSchnell,z100,nomtcp1\WObj:=BS_1606_1A;
MoveJ LHP_275,vSchnell,z100,nomtcp1\WObj:=BS_1606_1A;
MoveJ LHP_280, vSchnell, z100, nomtcp1\WObj:=BS_1606_1A;
MoveL LHP_285,vSchnell,z5,nomtcp1\WObj:=BS_1606_1A;
MoveL LHP_290,vSchnell,z5,nomtcp1\WObj:=BS_1606_1A;
MoveL LHP_295,vSchnell,z5,nomtcp1\WObj:=BS_1606_1A;
MoveL LHP_300,vSchnell,z5,nomtcp1\WObj:=BS_1606_1A;
MoveL LHP_305,vSchnell,z5,nomtcp1\WObj:=BS_1606_1A;
!
SpotL G0216190480BP20\VFO:=210\Vorhub_Auf, vSpot, nomtcp1\WObj:=BS_1606_1A;
!
MoveL LHP_310,vSchnell,z5,nomtcp1\WObj:=BS_1606_1A;
MoveL LHP_315,vSchnell,z5,nomtcp1\WObj:=BS_1606_1A;
MoveL LHP_320,vSchnell,z5,nomtcp1\WObj:=BS_1606_1A;
MoveL LHP_325,vSchnell,z5,nomtcp1\WObj:=BS_1606_1A;
MoveL LHP_330,vSchnell,z5,nomtcp1\WObj:=BS_1606_1A;
MoveL LHP_335,vSchnell,z5,nomtcp1\WObj:=BS_1606_1A;
MoveL LHP_340,vSchnell,z5,nomtcp1\WObj:=BS_1606_1A;
!
SpotL G0216022394BP20\VFO:=220\Vorhub_Auf,vSpot,nomtcp1\WObj:=BS_1606_1A;
!
MoveJ LHP_345, vSchnell, fine, nomtcp1\WObj:=BS_1606_1A;
!
!1606R04_1606R06
KOLLISION_ZONE 6\Freigabe;
!
MoveJ LHP_350, vSchnell, z100, nomtcp1\WObj:=BS_1606_1A;
!
SpotL G0216022386BP20\VFO:=210, vSpot, nomtcp1\WObj:=BS_1606_1A;
!
SpotL G0216047033BP20\VFO:=210,vSpot,nomtcp1\WObj:=BS_1606_1A;
!
SpotL G0216047032BP20\VFO:=210\Vorhub_Auf, vSpot, nomtcp1\WObj:=BS_1606_1A;
!
MoveJ LHP_355,vSchnell,z100,nomtcp1\WObj:=BS_1606_1A;
MoveJ LHP_360,vSchnell,z100,nomtcp1\WObj:=BS_1606_1A;
MoveJ LHP_365, vSchnell, z100, nomtcp1\WObj:=BS_1606_1A;
MoveJ LHP_370, vSchnell, z100, nomtcp1\WObj:=BS_1606_1A;
MoveJ LHP_375, vSchnell, z100, nomtcp1\WObj:=BS_1606_1A;
MoveJ LHP_380, vSchnell, z100, nomtcp1\WObj:=BS_1606_1A;
MoveJ LHP_385, vSchnell, z100, nomtcp1\WObj:=BS_1606_1A;
MoveJ LHP_390, vSchnell, fine, nomtcp1\WObj:=BS_1606_1A;
!
!1606R04_1606R06
KOLLISION_ZONE 7\Freigabe;
!
SpotL G0216190494BP20\VFO:=210,vSpot,nomtcp1\WObj:=BS_1606_1A;
!
SpotL G0216190496BP20\VFO:=210,vSpot,nomtcp1\WObj:=BS_1606_1A;
!
SpotL G0216190498BP20\VFO:=210,vSpot,nomtcp1\WObj:=BS_1606_1A;
!
MoveJ LHP_395,vSchnell,z100,nomtcp1\WObj:=BS_1606_1A;
!
SpotL G0216190488BP20\VFO:=210,vSpot,nomtcp1\WObj:=BS_1606_1A;
!
MoveJ LHP_400,vSchnell,z100,nomtcp1\WObj:=BS_1606_1A;
!
SpotL G0216190500BP20\VFO:=210\Vorhub_Auf,vSpot,nomtcp1\WObj:=BS_1606_1A;
!
MoveJ LHP_405,vSchnell,z100,nomtcp1\WObj:=BS_1606_1A;
MoveJ LHP_410,vSchnell,z100,nomtcp1\WObj:=BS_1606_1A;
MoveJ LHP_415,vSchnell,z100,nomtcp1\WObj:=BS_1606_1A;
MoveJ LHP_420,vSchnell,z100,nomtcp1\WObj:=BS_1606_1A;
MoveJ LHP_425,vSchnell,z100,nomtcp1\WObj:=BS_1606_1A;
MoveJ LHP_430,vSchnell,z100,nomtcp1\WObj:=BS_1606_1A;
MoveJ LHP_435,vSchnell,z100,nomtcp1\WObj:=BS_1606_1A;
!
SpotL G0216047028BP20\VFO:=210,vSpot,nomtcp1\WObj:=BS_1606_1A;
!
SpotL G0216047029BP20\VFO:=210,vSpot,nomtcp1\WObj:=BS_1606_1A;
!
SpotL G0216022368BP20\VFO:=210,vSpot,nomtcp1\WObj:=BS_1606_1A;
!
SpotL G0216022370BP20\VFO:=210\Vorhub_Auf,vSpot,nomtcp1\WObj:=BS_1606_1A;
!
MoveJ LHP_440, vSchnell, z100, nomtcp1\WObj:=BS_1606_1A;
MoveJ LHP_445, vSchnell, z100, nomtcp1\WObj:=BS_1606_1A;
MoveJ LHP_450, vSchnell, z100, nomtcp1\WObj:=BS_1606_1A;
MoveJ LHP_455, vSchnell, z100, nomtcp1\WObj:=BS_1606_1A;
MoveJ LHP_460, vSchnell, z100, nomtcp1\WObj:=BS_1606_1A;
MoveJ LHP_465, vSchnell, z100, nomtcp1\WObj:=BS_1606_1A;
!
SpotL G0216190436BP20\VFO:=210,vSpot,nomtcp1\WObj:=BS_1606_1A;
!
SpotL G0216190438BP20\VFO:=210,vSpot,nomtcp1\WObj:=BS_1606_1A;
!
SpotL G0216190440BP20\VFO:=210, vSpot, nomtcp1\WObj:=BS_1606_1A;
!
SpotL G0216023174BP20\VFO:=210,vSpot,nomtcp1\WObj:=BS_1606_1A;
!
SpotL G0216023172BP20\VFO:=210,vSpot,nomtcp1\WObj:=BS_1606_1A;
!
MoveJ LHP_470, vSchnell, fine, nomtcp1\WObj:=BS_1606_1A;
!
!1606R04_1606R06
KOLLISION_ZONE 8\Freigabe;
!
SpotL G0216023170BP20\VFO:=210,vSpot,nomtcp1\WObj:=BS_1606_1A;
!
SpotL G0216023168BP20\VFO:=210,vSpot,nomtcp1\WObj:=BS_1606_1A;
!
SpotL G0213195682BP20\VFO:=210,vSpot,nomtcp1\WObj:=BS_1606_1A;
!
SpotL G0213195680BP20\VFO:=210,vSpot,nomtcp1\WObj:=BS_1606_1A;
!
SpotL G0216190428BP20\VFO:=210,vSpot,nomtcp1\WObj:=BS_1606_1A;
!
SpotL G0216190430BP20\VFO:=210,vSpot,nomtcp1\WObj:=BS_1606_1A;
!
SpotL G0216190432BP20\VFO:=210,vSpot,nomtcp1\WObj:=BS_1606_1A;
!
SpotL G0216190434BP20\VFO:=210\Vorhub_Auf, vSpot, nomtcp1\WObj:=BS_1606_1A;
!
MoveJ LHP_475,vSchnell,z100,nomtcp1\WObj:=BS_1606_1A;
MoveJ LHP_480, vSchnell, z100, nomtcp1\WObj:=BS_1606_1A;
!
!
SpotL G0216190576BP20\VFO:=220,vSpot,nomtcp1\WObj:=BS_1606_1A;
!
SpotL G0213195678BP20\VFO:=210\Vorhub_Auf,vSpot,nomtcp1\WObj:=BS_1606_1A;
!
MoveJ LHP_485,vSchnell,z100,nomtcp1\WObj:=BS_1606_1A;
MoveJ LHP_490,vSchnell,z100,nomtcp1\WObj:=BS_1606_1A;
!
SpotL G0213195686BP20\VFO:=210,vSpot,nomtcp1\WObj:=BS_1606_1A;
!
SpotL G0213195688BP20\VFO:=210\Vorhub_Auf, vSpot, nomtcp1\WObj:=BS_1606_1A;
!
MoveJ LHP_495, vSchnell, z100, nomtcp1\WObj:=BS_1606_1A;
MoveJ LHP_500, vSchnell, z10, nomtcp1\WObj:=BS_1606_1A;
MoveJ LHP_505, vSchnell, z5, nomtcp1\WObj:=BS_1606_1A;
MoveJ LHP_510, vSchnell, z5, nomtcp1\WObj:=BS_1606_1A;
MoveJ LHP_515, vSchnell, z5, nomtcp1\WObj:=BS_1606_1A;
MoveJ LHP_520, vSchnell, z5, nomtcp1\WObj:=BS_1606_1A;
MoveJ LHP_525, vSchnell, z5, nomtcp1\WObj:=BS_1606_1A;
MoveJ LHP_530, vSchnell, fine, nomtcp1\WObj:=BS_1606_1A;
!
!1606R04_1606R06
KOLLISION_ZONE 1\Freigabe;
!
MoveJ LHP_535, vSchnell, z100, nomtcp1\WObj:=BS_1606_1A;
!
MoveJ ToolHome1,vSchnell,fine,nomtcp1;
!
!1606R04_1606R06
KOLLISION_ZONE 5\Freigabe;
!
ABL 254\ABL_WAIT;
ABL 255\ABL_SET;
!
!1606R04_1606R06
KOLLISION_ZONE 9\Anfrage;
!
!1606R04_1606R06
KOLLISION_ZONE 9\Freigabe;
!
ENDPROC



PROC swp_225500_0_st1606_1()

CONST robtarget LHP_000:=[[2573.53101,1238.19995,2660.84204],[0.56645757,-0.58473384,0.19941168,-0.54538715],[-1,-1,-1,4],[9E9,9E9,9E9,9E9,9E9,9E9]];
CONST robtarget LHP_005:=[[1933.57397,1076.34998,919.023987],[0.6739808,-0.04561597,0.22679393,-0.70159364],[-1,-1,-1,0],[9E9,9E9,9E9,9E9,9E9,9E9]];
CONST robtarget LHP_010:=[[1910.90503,994.687988,216.904999],[0.7042605,0.08468377,0.09847328,-0.6979605],[-1,-1,-1,0],[9E9,9E9,9E9,9E9,9E9,9E9]];
CONST robtarget LHP_015:=[[1910.89099,994.690002,-385.321991],[0.683501,0.087539785,0.09595496,-0.71830064],[-1,-1,-1,0],[9E9,9E9,9E9,9E9,9E9,9E9]];
CONST robtarget LHP_020:=[[1910.92,803.63,-358.65],[0.683496,0.087554,0.0959515,-0.718305],[-1,-1,-1,0],[9E+09,9E+09,9E+09,9E+09,9E+09,9E+09]];
CONST robtarget LHP_025:=[[1910.97,741.50,-281.66],[0.683494,0.0875455,0.0959486,-0.718307],[-1,-1,-1,0],[9E+09,9E+09,9E+09,9E+09,9E+09,9E+09]];
CONST robtarget LHP_030:=[[1910.91,559.83,-213.69],[0.686476,0.0613746,0.0695917,-0.721208],[-1,-1,-1,0],[9E+09,9E+09,9E+09,9E+09,9E+09,9E+09]];
CONST robtarget LHP_035:=[[1929.33,361.88,-170.13],[0.702471,0.0120548,-0.002609,-0.711605],[-1,0,-1,0],[9E+09,9E+09,9E+09,9E+09,9E+09,9E+09]];
CONST robtarget LHP_040:=[[2007.526,383.55899,-50.7519989],[0.75072795,0.000611088,0.00040383,-0.6606111],[-1,-1,-1,0],[9E9,9E9,9E9,9E9,9E9,9E9]];
CONST robtarget LHP_045:=[[1993.04797,313.046997,-31.7070007],[0.7336252,0.009941696,-0.001285905,-0.67948043],[-1,0,-1,0],[9E9,9E9,9E9,9E9,9E9,9E9]];
CONST robtarget LHP_050:=[[2002.59399,189.292999,-35.1940002],[0.73792726,0.009937888,-0.0012356,-0.67480594],[-1,0,-1,0],[9E9,9E9,9E9,9E9,9E9,9E9]];
CONST robtarget LHP_055:=[[1987.44,-5.82,-69.73],[0.747483,0.000551369,0.000433351,-0.664281],[-1,-1,-1,0],[9E+09,9E+09,9E+09,9E+09,9E+09,9E+09]];
CONST robtarget LHP_060:=[[1929.34,361.89,-170.15],[0.70247,0.0120598,-0.00260928,-0.711607],[-1,0,-1,0],[9E+09,9E+09,9E+09,9E+09,9E+09,9E+09]];
CONST robtarget LHP_065:=[[1910.91,559.85,-213.71],[0.686472,0.0613779,0.0695915,-0.721211],[-1,-1,-1,0],[9E+09,9E+09,9E+09,9E+09,9E+09,9E+09]];
CONST robtarget LHP_070:=[[1769.54,626.69,-228.36],[0.648406,0.063605,0.0595836,-0.756289],[-1,-1,-1,0],[9E+09,9E+09,9E+09,9E+09,9E+09,9E+09]];
CONST robtarget LHP_075:=[[1629.23,373.82,-175.88],[0.60566,0.011527,-0.00436593,-0.795628],[-1,0,-1,0],[9E+09,9E+09,9E+09,9E+09,9E+09,9E+09]];
CONST robtarget LHP_080:=[[1643.37,44.45,-93.67],[0.638426,0.0118697,-0.00343011,-0.769584],[-1,0,-1,0],[9E+09,9E+09,9E+09,9E+09,9E+09,9E+09]];
CONST robtarget LHP_085:=[[1645.79,51.65,-47.78],[0.621544,0.019299,-0.00963586,-0.783082],[-1,0,-1,0],[9E+09,9E+09,9E+09,9E+09,9E+09,9E+09]];
CONST robtarget LHP_090:=[[1652.62,133.53,-52.42],[0.605581,0.0130855,-0.00581803,-0.795655],[-1,0,-1,0],[9E+09,9E+09,9E+09,9E+09,9E+09,9E+09]];
CONST robtarget LHP_095:=[[1617.10803,350.912994,-180.268005],[0.56401443,0.037766688,0.053717423,-0.8231499],[-1,-1,-1,0],[9E9,9E9,9E9,9E9,9E9,9E9]];
CONST robtarget LHP_100:=[[1517.84,635.47,-254.71],[0.565141,-0.00404407,-0.00655324,-0.824958],[-1,0,-1,0],[9E+09,9E+09,9E+09,9E+09,9E+09,9E+09]];
CONST robtarget LHP_105:=[[1647.70,917.36,-357.05],[0.686537,0.012902,0.00966857,-0.726916],[-1,-1,-1,0],[9E+09,9E+09,9E+09,9E+09,9E+09,9E+09]];
CONST robtarget LHP_110:=[[1402.01,954.02,-347.18],[0.618002,-0.00350893,0.00682793,-0.786139],[-1,-1,-1,0],[9E+09,9E+09,9E+09,9E+09,9E+09,9E+09]];
CONST robtarget LHP_115:=[[1380.13,800.38,-342.28],[0.663576,-0.00391562,0.00660285,-0.74807],[-1,-1,-1,0],[9E+09,9E+09,9E+09,9E+09,9E+09,9E+09]];
CONST robtarget LHP_120:=[[1355.05,688.92,-230.68],[0.643458,-0.00406434,0.0069742,-0.765439],[-1,-1,-1,0],[9E+09,9E+09,9E+09,9E+09,9E+09,9E+09]];
CONST robtarget LHP_125:=[[1338.98,616.80,-217.15],[0.641931,-0.00377363,0.00673657,-0.766724],[-1,-1,-1,0],[9E+09,9E+09,9E+09,9E+09,9E+09,9E+09]];
CONST robtarget LHP_130:=[[1328.82,551.60,-198.45],[0.643236,-0.00380631,0.00669098,-0.765629],[-1,-1,-1,0],[9E+09,9E+09,9E+09,9E+09,9E+09,9E+09]];
CONST robtarget LHP_135:=[[1301.19,432.03,-200.08],[0.630965,0.0270779,0.0228783,-0.775001],[-1,-1,-1,0],[9E+09,9E+09,9E+09,9E+09,9E+09,9E+09]];
CONST robtarget LHP_140:=[[1315.22,418.75,-159.95],[0.640955,0.052567,0.0459758,-0.764395],[-1,-1,-1,0],[9E+09,9E+09,9E+09,9E+09,9E+09,9E+09]];
CONST robtarget LHP_145:=[[1314.89,402.01,-58.59],[0.643636,0.0406528,0.0359674,-0.763405],[-1,-1,-1,0],[9E+09,9E+09,9E+09,9E+09,9E+09,9E+09]];
CONST robtarget LHP_150:=[[1314.89,402.00,-58.59],[0.64363700,0.04065100,0.0359677,-0.7634040],[-1,-1,-1,0],[9E+09,9E+09,9E+09,9E+09,9E+09,9E+09]];
CONST robtarget LHP_155:=[[1315.25,418.75,-159.98],[0.640959,0.05257270,0.04597540,-0.7643910],[-1,-1,-1,0],[9E+09,9E+09,9E+09,9E+09,9E+09,9E+09]];
CONST robtarget LHP_160:=[[1301.20,432.03,-200.09],[0.630966,0.0270787,0.0228773,-0.775],[-1,-1,-1,0],[9E+09,9E+09,9E+09,9E+09,9E+09,9E+09]];
CONST robtarget LHP_165:=[[1328.84,551.60,-198.48],[0.643767,-0.00379566,0.00669219,-0.765183],[-1,-1,-1,0],[9E+09,9E+09,9E+09,9E+09,9E+09,9E+09]];
CONST robtarget LHP_170:=[[1356.81,663.69,-214.66],[0.64609,-0.00377796,0.00670482,-0.7632220],[-1,-1,-1,0],[9E+09,9E+09,9E+09,9E+09,9E+09,9E+09]];
CONST robtarget LHP_175:=[[1392.09,854.35,-337.39],[0.646086,-0.00378978,0.00670626,-0.763226],[-1,-1,-1,0],[9E+09,9E+09,9E+09,9E+09,9E+09,9E+09]];
CONST robtarget LHP_180:=[[1392.10,915.32,-339.98],[0.646085,-0.00379686,0.00670629,-0.763227],[-1,-1,-1,0],[9E+09,9E+09,9E+09,9E+09,9E+09,9E+09]];
CONST robtarget LHP_185:=[[1392.13,915.34,-336.92],[0.646086,-0.00378783,0.00670572,-0.763226],[-1,-1,-1,0],[9E+09,9E+09,9E+09,9E+09,9E+09,9E+09]];
CONST robtarget LHP_190:=[[1777.10,396.39,-174.51],[0.778298,0.00338922,-0.00251072,-0.62788],[-1,0,-1,0],[9E+09,9E+09,9E+09,9E+09,9E+09,9E+09]];
CONST robtarget LHP_195:=[[1816.72,397.75,-147.92],[0.816486,0.00152322,-0.000785194,-0.577362],[-1,0,-1,0],[9E+09,9E+09,9E+09,9E+09,9E+09,9E+09]];
CONST robtarget LHP_200:=[[1816.69,397.74,-147.92],[0.816487,0.00151316,-0.000780112,-0.577362],[-1,0,-1,0],[9E+09,9E+09,9E+09,9E+09,9E+09,9E+09]];
CONST robtarget LHP_205:=[[1684.99,383.29,-52.10],[0.598242,-0.000451381,-0.0146486,-0.801182],[-1,0,-1,0],[9E+09,9E+09,9E+09,9E+09,9E+09,9E+09]];
CONST robtarget LHP_210:=[[1517.37,845.68,-347.51],[0.603966,0.0765094,0.0409368,-0.792272],[-1,-1,-1,0],[9E+09,9E+09,9E+09,9E+09,9E+09,9E+09]];
CONST robtarget LHP_215:=[[1614.81,303.29,-114.97],[0.595541,4.37463E-06,7.52158E-05,-0.803325],[-1,-1,-1,0],[9E+09,9E+09,9E+09,9E+09,9E+09,9E+09]];
CONST robtarget LHP_220:=[[1496.10,381.00,-140.90],[0.501832,0.0142883,0.0357857,-0.864106],[-1,-1,-1,0],[9E+09,9E+09,9E+09,9E+09,9E+09,9E+09]];
CONST robtarget LHP_225:=[[1496.16,381.04,-179.37],[0.501836,0.0143261,0.0358019,-0.864103],[-1,-1,-1,0],[9E+09,9E+09,9E+09,9E+09,9E+09,9E+09]];
CONST robtarget LHP_230:=[[1517.37,556.59,-186.35],[0.545787,0.0365786,0.0545327,-0.835347],[-1,-1,-1,0],[9E+09,9E+09,9E+09,9E+09,9E+09,9E+09]];
CONST robtarget LHP_235:=[[1529.66,619.50,-150.47],[0.565262,-0.000227126,0.000165536,-0.824912],[-1,-1,-1,0],[9E+09,9E+09,9E+09,9E+09,9E+09,9E+09]];
CONST robtarget LHP_240:=[[1558.44,796.09,-349.49],[0.583985,0.0684408,0.0319346,-0.808244],[-1,-1,-1,0],[9E+09,9E+09,9E+09,9E+09,9E+09,9E+09]];
CONST robtarget LHP_245:=[[1477.93,985.71,-357.82],[0.551096,0.0897034,0.0519627,-0.827978],[-1,-1,-1,0],[9E+09,9E+09,9E+09,9E+09,9E+09,9E+09]];
CONST robtarget LHP_250:=[[807.86,896.51,-348.98],[0.475989,-0.019585,0.0486327,-0.877887],[-1,-1,-1,0],[9E+09,9E+09,9E+09,9E+09,9E+09,9E+09]];
CONST robtarget LHP_255:=[[807.84,813.89,-348.98],[0.47599,-0.0195894,0.0486332,-0.877887],[-1,-1,-1,0],[9E+09,9E+09,9E+09,9E+09,9E+09,9E+09]];
CONST robtarget LHP_260:=[[798.625,757.187988,-251.093002],[0.47488588,-0.019798715,0.048936285,-0.8784627],[-1,-1,-1,0],[9E9,9E9,9E9,9E9,9E9,9E9]];
CONST robtarget LHP_265:=[[687.672974,377.386993,-182.552002],[0.5034063,-0.04137853,0.03811411,-0.8622165],[-1,-1,-1,0],[9E9,9E9,9E9,9E9,9E9,9E9]];
CONST robtarget LHP_270:=[[796.06,403.61,2.12],[0.54967,-0.0809587,0.0198978,-0.831212],[-1,-1,-1,0],[9E+09,9E+09,9E+09,9E+09,9E+09,9E+09]];
CONST robtarget LHP_275:=[[951.56,404.05,-36.64],[0.666081,-0.0483269,0.018538,-0.744081],[-1,-1,-1,0],[9E+09,9E+09,9E+09,9E+09,9E+09,9E+09]];
CONST robtarget LHP_280:=[[1053.17,384.08,-147.35],[0.741703,0.0276666,0.0554714,-0.667858],[-1,-1,-1,0],[9E+09,9E+09,9E+09,9E+09,9E+09,9E+09]];
CONST robtarget LHP_285:=[[1117.00,437.68,-186.63],[0.764604,0.0628167,0.0737039,-0.637183],[-1,-1,-1,0],[9E+09,9E+09,9E+09,9E+09,9E+09,9E+09]];
CONST robtarget LHP_290:=[[1206.43,437.70,-186.66],[0.808318,0.0679399,0.0690137,-0.580726],[-1,-1,-1,0],[9E+09,9E+09,9E+09,9E+09,9E+09,9E+09]];
CONST robtarget LHP_295:=[[1254.01,306.17,-147.47],[0.819239,0.0692406,0.0677067,-0.565215],[-1,-1,-1,0],[9E+09,9E+09,9E+09,9E+09,9E+09,9E+09]];
CONST robtarget LHP_300:=[[1294.76,251.64,-118.31],[0.839473,0.0657832,0.0563212,-0.536456],[-1,-1,-1,0],[9E+09,9E+09,9E+09,9E+09,9E+09,9E+09]];
CONST robtarget LHP_305:=[[1302.68,268.91,-77.08],[0.850295,0.0194976,0.0312356,-0.525017],[-1,-1,-1,0],[9E+09,9E+09,9E+09,9E+09,9E+09,9E+09]];
CONST robtarget LHP_310:=[[1302.67,268.92,-77.09],[0.850295,0.0194964,0.0312402,-0.525016],[-1,-1,-1,0],[9E+09,9E+09,9E+09,9E+09,9E+09,9E+09]];
CONST robtarget LHP_315:=[[1294.76,251.64,-118.31],[0.839473,0.0657839,0.0563209,-0.536456],[-1,-1,-1,0],[9E+09,9E+09,9E+09,9E+09,9E+09,9E+09]];
CONST robtarget LHP_320:=[[1254.01,306.17,-147.47],[0.819239,0.0692405,0.0677067,-0.565215],[-1,-1,-1,0],[9E+09,9E+09,9E+09,9E+09,9E+09,9E+09]];
CONST robtarget LHP_325:=[[1206.43,437.70,-186.66],[0.808318,0.0679399,0.0690137,-0.580726],[-1,-1,-1,0],[9E+09,9E+09,9E+09,9E+09,9E+09,9E+09]];
CONST robtarget LHP_330:=[[1117.00,437.68,-186.63],[0.764604,0.0628167,0.0737039,-0.637183],[-1,-1,-1,0],[9E+09,9E+09,9E+09,9E+09,9E+09,9E+09]];
CONST robtarget LHP_335:=[[1116.98,404.12,-155.12],[0.767929,0.0632076,0.0733697,-0.633172],[-1,-1,-1,0],[9E+09,9E+09,9E+09,9E+09,9E+09,9E+09]];
CONST robtarget LHP_340:=[[1116.98,404.12,-77.86],[0.763388,0.0288222,0.0341692,-0.644392],[-1,-1,-1,0],[9E+09,9E+09,9E+09,9E+09,9E+09,9E+09]];
CONST robtarget LHP_345:=[[951.56,404.05,-36.63],[0.666079,-0.0483271,0.018537,-0.744083],[-1,-1,-1,0],[9E+09,9E+09,9E+09,9E+09,9E+09,9E+09]];
CONST robtarget LHP_350:=[[863.42,413.34,0.81],[0.590286,-0.0726155,0.0279581,-0.803435],[-1,-1,-1,0],[9E+09,9E+09,9E+09,9E+09,9E+09,9E+09]];
CONST robtarget LHP_355:=[[687.66803,377.371002,-182.531006],[0.5034058,-0.04138605,0.0381097,-0.8622166],[-1,-1,-1,0],[9E9,9E9,9E9,9E9,9E9,9E9]];
CONST robtarget LHP_360:=[[798.580994,757.198975,-251.070007],[0.47486982,-0.019813199,0.04892835,-0.8784715],[-1,-1,-1,0],[9E9,9E9,9E9,9E9,9E9,9E9]];
CONST robtarget LHP_365:=[[961.40,981.11,-456.97],[0.440335,0.0935079,0.0750373,-0.889792],[-1,-1,-1,0],[9E+09,9E+09,9E+09,9E+09,9E+09,9E+09]];
CONST robtarget LHP_370:=[[1477.90,985.72,-357.83],[0.558631,0.0901634,0.0511329,-0.822914],[-1,-1,-1,0],[9E+09,9E+09,9E+09,9E+09,9E+09,9E+09]];
CONST robtarget LHP_375:=[[1538.22,786.86,-339.64],[0.544053,0.0691445,0.0535195,-0.834482],[-1,-1,-1,0],[9E+09,9E+09,9E+09,9E+09,9E+09,9E+09]];
CONST robtarget LHP_380:=[[1502.92,670.32,-266.02],[0.529086,0.0479959,0.0506422,-0.845695],[-1,-1,-1,0],[9E+09,9E+09,9E+09,9E+09,9E+09,9E+09]];
CONST robtarget LHP_385:=[[1496.13,395.81,-167.92],[0.501832,0.0142997,0.0357903,-0.864106],[-1,-1,-1,0],[9E+09,9E+09,9E+09,9E+09,9E+09,9E+09]];
CONST robtarget LHP_390:=[[1515.01,305.29,-41.45],[0.500229,-6.95049E-05,2.93455E-05,-0.865893],[-1,-1,-1,0],[9E+09,9E+09,9E+09,9E+09,9E+09,9E+09]];
CONST robtarget LHP_395:=[[1371.85706,156.694901,-47.4344292],[0.4850808,-0.004593692,-0.00611278,-0.8744359],[-1,0,-1,0],[9E9,9E9,9E9,9E9,9E9,9E9]];
CONST robtarget LHP_400:=[[1371.81006,156.684998,-41.7470016],[0.48507392,-0.004586132,-0.006106427,-0.8744398],[-1,0,-1,0],[9E9,9E9,9E9,9E9,9E9,9E9]];
CONST robtarget LHP_405:=[[1492.72,315.84,-138.22],[0.571745,-0.00395765,-0.00657566,-0.820395],[-1,0,-1,0],[9E+09,9E+09,9E+09,9E+09,9E+09,9E+09]];
CONST robtarget LHP_410:=[[1568.64,542.95,-202.94],[0.571744,-0.00395848,-0.00658119,-0.820396],[-1,0,-1,0],[9E+09,9E+09,9E+09,9E+09,9E+09,9E+09]];
CONST robtarget LHP_415:=[[1568.58,736.45,-284.14],[0.571745,-0.00397095,-0.00657964,-0.820396],[-1,0,-1,0],[9E+09,9E+09,9E+09,9E+09,9E+09,9E+09]];
CONST robtarget LHP_420:=[[1508.30,917.00,-395.22],[0.556499,0.0508994,0.0317793,-0.828678],[-1,-1,-1,0],[9E+09,9E+09,9E+09,9E+09,9E+09,9E+09]];
CONST robtarget LHP_425:=[[1495.25,987.39,-357.83],[0.551104,0.0895725,0.0518729,-0.827992],[-1,-1,-1,0],[9E+09,9E+09,9E+09,9E+09,9E+09,9E+09]];
CONST robtarget LHP_430:=[[1328.35,635.44,-278.20],[0.501405,0.0212305,0.11734,-0.856956],[-1,-1,0,0],[9E+09,9E+09,9E+09,9E+09,9E+09,9E+09]];
CONST robtarget LHP_435:=[[1126.70,526.89,-238.13],[0.384755,0.0646485,0.107006,-0.914513],[-1,-1,0,0],[9E+09,9E+09,9E+09,9E+09,9E+09,9E+09]];
CONST robtarget LHP_440:=[[1126.70,526.87,-238.14],[0.384757,0.0646487,0.107006,-0.914512],[-1,-1,0,0],[9E+09,9E+09,9E+09,9E+09,9E+09,9E+09]];
CONST robtarget LHP_445:=[[1328.35,635.43,-278.21],[0.501406,0.0212292,0.11734,-0.856956],[-1,-1,0,0],[9E+09,9E+09,9E+09,9E+09,9E+09,9E+09]];
CONST robtarget LHP_450:=[[1495.26,987.39,-357.84],[0.551103,0.0895724,0.0518701,-0.827993],[-1,-1,-1,0],[9E+09,9E+09,9E+09,9E+09,9E+09,9E+09]];
CONST robtarget LHP_455:=[[1606.25,805.30,-336.47],[0.591189,0.0705667,0.0504833,-0.801852],[-1,-1,-1,0],[9E+09,9E+09,9E+09,9E+09,9E+09,9E+09]];
CONST robtarget LHP_460:=[[1846.21,646.41,-266.45],[0.66313,0.055392,0.0578373,-0.744207],[-1,-1,-1,0],[9E+09,9E+09,9E+09,9E+09,9E+09,9E+09]];
CONST robtarget LHP_465:=[[1831.93,634.62,-78.38],[0.625946,0.00957367,0.0100376,-0.779743],[-1,-1,-1,0],[9E+09,9E+09,9E+09,9E+09,9E+09,9E+09]];
CONST robtarget LHP_470:=[[1793.13,513.60,-41.97],[0.578209,9.78811E-06,-2.13769E-07,-0.815889],[-1,-1,-1,0],[9E+09,9E+09,9E+09,9E+09,9E+09,9E+09]];
CONST robtarget LHP_475:=[[1581.22,548.75,-125.86],[0.508525,0.0149425,0.00198371,-0.860915],[-1,0,-1,0],[9E+09,9E+09,9E+09,9E+09,9E+09,9E+09]];
CONST robtarget LHP_480:=[[1526.71,530.36,-111.44],[0.495097,0.0157343,0.00230728,-0.868692],[-1,0,-1,0],[9E+09,9E+09,9E+09,9E+09,9E+09,9E+09]];
CONST robtarget LHP_485:=[[1496.52905,533.620972,-169.427002],[0.5015252,0.014323151,0.035049833,-0.8643141],[-1,-1,-1,0],[9E9,9E9,9E9,9E9,9E9,9E9]];
CONST robtarget LHP_490:=[[1628.88,359.00,-167.42],[0.509965,0.00587853,-0.00326077,-0.860169],[-1,0,-1,0],[9E+09,9E+09,9E+09,9E+09,9E+09,9E+09]];
CONST robtarget LHP_495:=[[1653.10,363.04,-167.43],[0.50985,0.0307676,0.0114918,-0.859636],[-1,0,-1,0],[9E+09,9E+09,9E+09,9E+09,9E+09,9E+09]];
CONST robtarget LHP_500:=[[1734.14,581.56,-229.81],[0.51369,0.0926739,0.046858,-0.851668],[-1,-1,-1,0],[9E+09,9E+09,9E+09,9E+09,9E+09,9E+09]];
CONST robtarget LHP_505:=[[1850.77,754.32,-287.10],[0.562259,0.138379,0.0973397,-0.809469],[-1,-1,-1,0],[9E+09,9E+09,9E+09,9E+09,9E+09,9E+09]];
CONST robtarget LHP_510:=[[1850.71,883.30,-361.37],[0.589549,0.148661,0.155296,-0.778598],[-1,-1,-1,0],[9E+09,9E+09,9E+09,9E+09,9E+09,9E+09]];
CONST robtarget LHP_515:=[[1850.60,911.16,-304.76],[0.610795,0.143869,0.202267,-0.751877],[-1,-1,-1,0],[9E+09,9E+09,9E+09,9E+09,9E+09,9E+09]];
CONST robtarget LHP_520:=[[1845.93,938.54,-187.19],[0.617535,0.126482,0.223985,-0.743292],[-1,-1,-1,0],[9E+09,9E+09,9E+09,9E+09,9E+09,9E+09]];
CONST robtarget LHP_525:=[[1839.91,764.25,251.37],[0.609113,0.0794277,0.135403,-0.777392],[-1,-1,-1,0],[9E+09,9E+09,9E+09,9E+09,9E+09,9E+09]];
CONST robtarget LHP_530:=[[1951.53,815.35,1215.32],[0.610126,-0.0704393,-0.00824645,-0.789124],[-1,0,-1,0],[9E+09,9E+09,9E+09,9E+09,9E+09,9E+09]];
CONST robtarget LHP_535:=[[2438.93,960.39,2235.39],[0.671457,-0.189483,-0.125804,-0.705277],[-1,0,-1,0],[9E+09,9E+09,9E+09,9E+09,9E+09,9E+09]];
!provisorische Punkte f?r SP-Versetzung in Zone2
CONST robtarget LHP_605:=[[1647.70,917.36,-357.05],[0.686537,0.012902,0.00966857,-0.726916],[-1,-1,-1,0],[9E+09,9E+09,9E+09,9E+09,9E+09,9E+09]];
CONST robtarget LHP_610:=[[1620.32,602.14,-205.68],[0.637115,0.00115264,-0.000310519,-0.770768],[-1,0,-1,0],[9E+09,9E+09,9E+09,9E+09,9E+09,9E+09]];
CONST robtarget LHP_620:=[[1912.93,601.14,-205.68],[0.710988,0.0011134,-0.000423279,-0.703204],[-1,0,-1,0],[9E+09,9E+09,9E+09,9E+09,9E+09,9E+09]];
CONST robtarget LHP_625:=[[1919.94,393.08,-177.19],[0.710987,0.00110842,-0.000423915,-0.703204],[-1,0,-1,0],[9E+09,9E+09,9E+09,9E+09,9E+09,9E+09]];
CONST robtarget LHP_630:=[[1919.96,393.09,-177.22],[0.710988,0.0011168,-0.000424803,-0.703203],[-1,0,-1,0],[9E+09,9E+09,9E+09,9E+09,9E+09,9E+09]];
CONST robtarget LHP_635:=[[1912.96,653.53,-205.68],[0.710987,0.00111256,-0.000425587,-0.703204],[-1,0,-1,0],[9E+09,9E+09,9E+09,9E+09,9E+09,9E+09]];
CONST robtarget LHP_600:=[[1990.20,974.03,1486.76],[0.667207,-0.21865,0.214527,-0.678974],[-1,-1,-1,0],[9E+09,9E+09,9E+09,9E+09,9E+09,9E+09]];
! ------------------------------------------------------------
! Unterprogramm:
! Stand
! Daimler AG - Werk Ludwigsfelde
! ------------------------------------------------------------
! ************************************************************
! Kommentar: Achtung
! automatisch generiert!!!!!!!!!!!!!!!!!!
! ************************************************************

! Robotername: 1606R04
! Anlagenbezeichn: Linie 16 Stations-Nr: 1606
! Stand / Version: 04.08.2009 / 1.1
! Name Bearbeiter: Karmann
! Applikationssteuerung: Punktschweissen
! Baumuster: FHL T1 R2


INIT_SW_BASE;

WKZ_1_AUFNEHMEN;
!
MoveJ ToolHome1,vSchnell,fine,nomtcp1;
!
MoveJ LHP_000,vSchnell,fine,nomtcp1\WObj:=BS_1606_1A;
!
Vorhub\auf;
!
ABL 2\ABL_WAIT;
!
ABL 10\ABL_SET;

